LIN {X -0.118,Y -195.849,Z 1330.705,A 0.000,B 0.000,C 90.000,E1 126.870} C_DIS
LIN {X 0.022,Y -199.211,Z 1330.695,A 0.000,B 0.000,C 90.000,E1 125.105} C_DIS
LIN {X -0.016,Y -309.077,Z 1330.695,A 0.000,B 0.000,C 90.000,E1 125.105} C_DIS
LIN {X -0.170,Y -310.750,Z 1330.695,A 0.000,B 0.000,C 90.000,E1 125.105} C_DIS
LIN {X 0.024,Y -314.683,Z 1330.694,A 0.000,B 0.000,C 90.000,E1 124.898} C_DIS
LIN {X -0.037,Y -316.948,Z 1330.693,A 0.000,B 0.000,C 90.000,E1 124.739} C_DIS
LIN {X -0.082,Y -320.065,Z 1330.691,A 0.000,B 0.000,C 90.000,E1 124.405} C_DIS
LIN {X -0.155,Y -322.032,Z 1330.689,A 0.000,B 0.000,C 90.000,E1 124.119} C_DIS
LIN {X 0.038,Y -323.567,Z 1330.688,A 0.000,B 0.000,C 90.000,E1 123.785} C_DIS
LIN {X -0.056,Y -325.946,Z 1330.684,A 0.000,B 0.000,C 90.000,E1 123.166} C_DIS
LIN {X -0.055,Y -336.432,Z 1330.668,A 0.000,B 0.000,C 90.000,E1 120.335} C_DIS
LIN {X 0.200,Y -348.268,Z 1330.653,A 0.000,B 0.000,C 90.000,E1 117.513} C_DIS
LIN {X 0.001,Y -361.549,Z 1330.638,A 0.000,B 0.000,C 90.000,E1 114.823} C_DIS
LIN {X -0.050,Y -374.665,Z 1330.625,A 0.000,B 0.000,C 90.000,E1 112.461} C_DIS
LIN {X 0.093,Y -389.108,Z 1330.612,A 0.000,B 0.000,C 90.000,E1 110.120} C_DIS
LIN {X -0.043,Y -404.981,Z 1330.599,A 0.000,B 0.000,C 90.000,E1 107.873} C_DIS
LIN {X -0.042,Y -422.391,Z 1330.587,A 0.000,B 0.000,C 90.000,E1 105.662} C_DIS
LIN {X -0.232,Y -441.441,Z 1330.575,A 0.000,B 0.000,C 90.000,E1 103.536} C_DIS
LIN {X 0.089,Y -461.498,Z 1330.564,A 0.000,B 0.000,C 90.000,E1 101.478} C_DIS
LIN {X 0.089,Y -479.451,Z 1330.555,A 0.000,B 0.000,C 90.000,E1 99.849} C_DIS
LIN {X 0.151,Y -481.477,Z 1330.553,A 0.000,B 0.000,C 90.000,E1 99.613} C_DIS
LIN {X 0.212,Y -483.021,Z 1330.552,A 0.000,B 0.000,C 90.000,E1 99.378} C_DIS
LIN {X 0.017,Y -484.300,Z 1330.551,A 0.000,B 0.000,C 90.000,E1 99.151} C_DIS
LIN {X -0.100,Y -485.240,Z 1330.549,A 0.000,B 0.000,C 90.000,E1 98.916} C_DIS
LIN {X 0.086,Y -486.268,Z 1330.547,A 0.000,B 0.000,C 90.000,E1 98.398} C_DIS
LIN {X -0.202,Y -486.295,Z 1330.544,A 0.000,B 0.000,C 90.000,E1 97.936} C_DIS
LIN {X 0.062,Y -485.327,Z 1330.541,A 0.000,B 0.000,C 90.000,E1 97.409} C_DIS
LIN {X -0.220,Y -483.199,Z 1330.538,A 0.000,B 0.000,C 90.000,E1 96.947} C_DIS
LIN {X 0.088,Y -481.557,Z 1330.537,A 0.000,B 0.000,C 90.000,E1 96.663} C_DIS
LIN {X 0.091,Y -470.630,Z 1330.529,A 0.000,B 0.000,C 90.000,E1 95.163} C_DIS
LIN {X -0.105,Y -457.075,Z 1330.517,A 0.000,B 0.000,C 90.000,E1 93.154} C_DIS
LIN {X 0.043,Y -442.213,Z 1330.505,A 0.000,B 0.000,C 90.000,E1 90.802} C_DIS
LIN {X 0.074,Y -425.766,Z 1330.488,A 0.000,B 0.000,C 90.000,E1 87.879} C_DIS
LIN {X 0.057,Y -415.709,Z 1330.478,A 0.000,B 0.000,C 90.000,E1 85.988} C_DIS
LIN {X -0.119,Y -405.430,Z 1330.467,A 0.000,B 0.000,C 90.000,E1 84.090} C_DIS
LIN {X -0.079,Y -396.463,Z 1330.458,A 0.000,B 0.000,C 90.000,E1 82.413} C_DIS
LIN {X -0.194,Y -387.225,Z 1330.448,A 0.000,B 0.000,C 90.000,E1 80.735} C_DIS
LIN {X -0.039,Y -377.786,Z 1330.439,A 0.000,B 0.000,C 90.000,E1 78.993} C_DIS
LIN {X 0.079,Y -366.465,Z 1330.427,A 0.000,B 0.000,C 90.000,E1 76.937} C_DIS
LIN {X 0.042,Y -354.979,Z 1330.416,A 0.000,B 0.000,C 90.000,E1 74.866} C_DIS
LIN {X -0.132,Y -343.438,Z 1330.404,A 0.000,B 0.000,C 90.000,E1 72.779} C_DIS
LIN {X -0.041,Y -330.180,Z 1330.391,A 0.000,B 0.000,C 90.000,E1 70.296} C_DIS
LIN {X -0.165,Y -317.253,Z 1330.376,A 0.000,B 0.000,C 90.000,E1 67.794} C_DIS
LIN {X -0.017,Y -300.759,Z 1330.357,A 0.000,B 0.000,C 90.000,E1 64.204} C_DIS
LIN {X -0.088,Y -291.482,Z 1330.344,A 0.000,B 0.000,C 90.000,E1 61.897} C_DIS
LIN {X -0.060,Y -284.436,Z 1330.333,A 0.000,B 0.000,C 90.000,E1 59.871} C_DIS
LIN {X 0.090,Y -274.075,Z 1330.314,A 0.000,B 0.000,C 90.000,E1 56.421} C_DIS
LIN {X -0.062,Y -264.729,Z 1330.294,A 0.000,B 0.000,C 90.000,E1 52.970} C_DIS
LIN {X 0.136,Y -255.963,Z 1330.275,A 0.000,B 0.000,C 90.000,E1 49.380} C_DIS
LIN {X -0.041,Y -249.331,Z 1330.259,A 0.000,B 0.000,C 90.000,E1 46.539} C_DIS
LIN {X 0.104,Y -241.390,Z 1330.238,A 0.000,B 0.000,C 90.000,E1 42.852} C_DIS
LIN {X -0.129,Y -234.080,Z 1330.218,A 0.000,B 0.000,C 90.000,E1 39.197} C_DIS
LIN {X 0.032,Y -227.630,Z 1330.197,A 0.000,B 0.000,C 90.000,E1 35.391} C_DIS
LIN {X -0.031,Y -222.216,Z 1330.175,A 0.000,B 0.000,C 90.000,E1 31.592} C_DIS
LIN {X 0.009,Y -217.022,Z 1330.150,A 0.000,B 0.000,C 90.000,E1 26.950} C_DIS
LIN {X -0.033,Y -212.863,Z 1330.124,A 0.000,B 0.000,C 90.000,E1 22.280} C_DIS
LIN {X -0.082,Y -209.866,Z 1330.102,A 0.000,B 0.000,C 90.000,E1 18.362} C_DIS
LIN {X -0.046,Y -207.669,Z 1330.084,A 0.000,B 0.000,C 90.000,E1 15.190} C_DIS
LIN {X -0.028,Y -205.583,Z 1330.067,A 0.000,B 0.000,C 90.000,E1 12.007} C_DIS
LIN {X -0.090,Y -202.497,Z 1330.036,A 0.000,B 0.000,C 90.000,E1 6.429} C_DIS
LIN {X 0.000,Y -200.364,Z 1330.000,A 0.000,B 0.000,C 90.000,E1 360.000} C_DIS
LIN {X 0.070,Y -200.097,Z 1329.962,A 0.000,B 0.000,C 90.000,E1 353.053} C_DIS
LIN {X -0.087,Y -201.859,Z 1329.926,A 0.000,B 0.000,C 90.000,E1 346.645} C_DIS
LIN {X 0.053,Y -205.124,Z 1329.894,A 0.000,B 0.000,C 90.000,E1 340.986} C_DIS
LIN {X -0.036,Y -209.391,Z 1329.868,A 0.000,B 0.000,C 90.000,E1 336.230} C_DIS
LIN {X -0.037,Y -213.991,Z 1329.846,A 0.000,B 0.000,C 90.000,E1 332.281} C_DIS
LIN {X 0.135,Y -219.620,Z 1329.824,A 0.000,B 0.000,C 90.000,E1 328.329} C_DIS
LIN {X 0.086,Y -226.283,Z 1329.803,A 0.000,B 0.000,C 90.000,E1 324.482} C_DIS
LIN {X -0.004,Y -232.326,Z 1329.786,A 0.000,B 0.000,C 90.000,E1 321.457} C_DIS
LIN {X -0.064,Y -240.993,Z 1329.765,A 0.000,B 0.000,C 90.000,E1 317.715} C_DIS
LIN {X 0.112,Y -249.732,Z 1329.747,A 0.000,B 0.000,C 90.000,E1 314.352} C_DIS
LIN {X 0.033,Y -258.740,Z 1329.730,A 0.000,B 0.000,C 90.000,E1 311.472} C_DIS
LIN {X -0.027,Y -267.675,Z 1329.717,A 0.000,B 0.000,C 90.000,E1 308.991} C_DIS
LIN {X 0.091,Y -279.387,Z 1329.701,A 0.000,B 0.000,C 90.000,E1 306.171} C_DIS
LIN {X 0.074,Y -289.324,Z 1329.690,A 0.000,B 0.000,C 90.000,E1 304.119} C_DIS
LIN {X -0.087,Y -298.444,Z 1329.680,A 0.000,B 0.000,C 90.000,E1 302.467} C_DIS
LIN {X -0.017,Y -308.572,Z 1329.671,A 0.000,B 0.000,C 90.000,E1 300.797} C_DIS
LIN {X 0.008,Y -317.490,Z 1329.664,A 0.000,B 0.000,C 90.000,E1 299.489} C_DIS
LIN {X -0.020,Y -329.613,Z 1329.655,A 0.000,B 0.000,C 90.000,E1 297.897} C_DIS
LIN {X 0.065,Y -350.580,Z 1329.641,A 0.000,B 0.000,C 90.000,E1 295.412} C_DIS
LIN {X -0.084,Y -363.624,Z 1329.633,A 0.000,B 0.000,C 90.000,E1 293.951} C_DIS
LIN {X 0.018,Y -373.873,Z 1329.626,A 0.000,B 0.000,C 90.000,E1 292.770} C_DIS
LIN {X 0.120,Y -383.899,Z 1329.620,A 0.000,B 0.000,C 90.000,E1 291.589} C_DIS
LIN {X -0.166,Y -400.941,Z 1329.609,A 0.000,B 0.000,C 90.000,E1 289.631} C_DIS
LIN {X -0.083,Y -415.751,Z 1329.600,A 0.000,B 0.000,C 90.000,E1 287.946} C_DIS
LIN {X -0.142,Y -425.351,Z 1329.594,A 0.000,B 0.000,C 90.000,E1 286.858} C_DIS
LIN {X 0.029,Y -432.158,Z 1329.589,A 0.000,B 0.000,C 90.000,E1 286.024} C_DIS
LIN {X -0.149,Y -438.442,Z 1329.585,A 0.000,B 0.000,C 90.000,E1 285.245} C_DIS
LIN {X 0.034,Y -444.085,Z 1329.580,A 0.000,B 0.000,C 90.000,E1 284.426} C_DIS
LIN {X -0.044,Y -449.062,Z 1329.576,A 0.000,B 0.000,C 90.000,E1 283.647} C_DIS
LIN {X -0.196,Y -453.340,Z 1329.571,A 0.000,B 0.000,C 90.000,E1 282.883} C_DIS
LIN {X 0.140,Y -456.820,Z 1329.567,A 0.000,B 0.000,C 90.000,E1 282.063} C_DIS
LIN {X -0.041,Y -457.839,Z 1329.566,A 0.000,B 0.000,C 90.000,E1 281.827} C_DIS
LIN {X 0.057,Y -459.565,Z 1329.563,A 0.000,B 0.000,C 90.000,E1 281.299} C_DIS
LIN {X 0.074,Y -460.955,Z 1329.560,A 0.000,B 0.000,C 90.000,E1 280.782} C_DIS
LIN {X 0.189,Y -461.962,Z 1329.557,A 0.000,B 0.000,C 90.000,E1 280.254} C_DIS
LIN {X -0.146,Y -462.526,Z 1329.554,A 0.000,B 0.000,C 90.000,E1 279.782} C_DIS
LIN {X -0.099,Y -462.700,Z 1329.551,A 0.000,B 0.000,C 90.000,E1 279.265} C_DIS
LIN {X -0.044,Y -462.433,Z 1329.549,A 0.000,B 0.000,C 90.000,E1 278.746} C_DIS
LIN {X 0.080,Y -461.733,Z 1329.546,A 0.000,B 0.000,C 90.000,E1 278.219} C_DIS
LIN {X 0.135,Y -460.499,Z 1329.543,A 0.000,B 0.000,C 90.000,E1 277.701} C_DIS
LIN {X 0.011,Y -457.672,Z 1329.539,A 0.000,B 0.000,C 90.000,E1 276.947} C_DIS
LIN {X 0.047,Y -455.107,Z 1329.536,A 0.000,B 0.000,C 90.000,E1 276.429} C_DIS
LIN {X -0.189,Y -453.660,Z 1329.534,A 0.000,B 0.000,C 90.000,E1 276.201} C_DIS
LIN {X -0.173,Y -450.230,Z 1329.531,A 0.000,B 0.000,C 90.000,E1 275.682} C_DIS
LIN {X -0.175,Y -446.094,Z 1329.529,A 0.000,B 0.000,C 90.000,E1 275.163} C_DIS
LIN {X 0.015,Y -443.722,Z 1329.527,A 0.000,B 0.000,C 90.000,E1 274.878} C_DIS
LIN {X 0.079,Y -438.319,Z 1329.524,A 0.000,B 0.000,C 90.000,E1 274.359} C_DIS
LIN {X -0.025,Y -432.416,Z 1329.522,A 0.000,B 0.000,C 90.000,E1 273.898} C_DIS
LIN {X -0.196,Y -426.155,Z 1329.519,A 0.000,B 0.000,C 90.000,E1 273.498} C_DIS
LIN {X 0.037,Y -419.659,Z 1329.517,A 0.000,B 0.000,C 90.000,E1 273.094} C_DIS
LIN {X 0.156,Y -413.002,Z 1329.515,A 0.000,B 0.000,C 90.000,E1 272.751} C_DIS
LIN {X 0.139,Y -406.290,Z 1329.514,A 0.000,B 0.000,C 90.000,E1 272.465} C_DIS
LIN {X -0.014,Y -399.093,Z 1329.512,A 0.000,B 0.000,C 90.000,E1 272.236} C_DIS
LIN {X 0.119,Y -391.578,Z 1329.511,A 0.000,B 0.000,C 90.000,E1 272.007} C_DIS
LIN {X 0.130,Y -383.979,Z 1329.510,A 0.000,B 0.000,C 90.000,E1 271.835} C_DIS
LIN {X -0.002,Y -376.274,Z 1329.510,A 0.000,B 0.000,C 90.000,E1 271.718} C_DIS
LIN {X 0.034,Y -367.410,Z 1329.509,A 0.000,B 0.000,C 90.000,E1 271.604} C_DIS
LIN {X -0.025,Y -358.395,Z 1329.509,A 0.000,B 0.000,C 90.000,E1 271.547} C_DIS
LIN {X 0.157,Y -350.749,Z 1329.508,A 0.000,B 0.000,C 90.000,E1 271.489} C_DIS
LIN {X 0.052,Y -181.350,Z 1329.508,A 0.000,B 0.000,C 90.000,E1 271.489} C_DIS
LIN {X -0.083,Y -181.556,Z 1329.500,A 0.000,B 0.000,C 90.000,E1 270.000} C_DIS
LIN {X 0.054,Y -180.901,Z 1329.474,A 0.000,B 0.000,C 90.000,E1 265.241} C_DIS
LIN {X 0.003,Y -180.225,Z 1329.464,A 0.000,B 0.000,C 90.000,E1 263.571} C_DIS
LIN {X -0.044,Y -179.040,Z 1329.446,A 0.000,B 0.000,C 90.000,E1 260.208} C_DIS
LIN {X 0.020,Y -178.707,Z 1329.441,A 0.000,B 0.000,C 90.000,E1 259.342} C_DIS
LIN {X -0.039,Y -175.755,Z 1329.412,A 0.000,B 0.000,C 90.000,E1 254.267} C_DIS
LIN {X -0.037,Y -171.938,Z 1329.384,A 0.000,B 0.000,C 90.000,E1 249.135} C_DIS
LIN {X -0.061,Y -171.321,Z 1329.379,A 0.000,B 0.000,C 90.000,E1 248.284} C_DIS
LIN {X -0.008,Y -167.578,Z 1329.355,A 0.000,B 0.000,C 90.000,E1 243.948} C_DIS
LIN {X -0.068,Y -166.211,Z 1329.346,A 0.000,B 0.000,C 90.000,E1 242.231} C_DIS
LIN {X -0.080,Y -162.975,Z 1329.326,A 0.000,B 0.000,C 90.000,E1 238.742} C_DIS
LIN {X -0.032,Y -160.889,Z 1329.312,A 0.000,B 0.000,C 90.000,E1 236.087} C_DIS
LIN {X -0.054,Y -157.658,Z 1329.292,A 0.000,B 0.000,C 90.000,E1 232.557} C_DIS
LIN {X 0.004,Y -155.696,Z 1329.277,A 0.000,B 0.000,C 90.000,E1 229.865} C_DIS
LIN {X -0.060,Y -151.960,Z 1329.252,A 0.000,B 0.000,C 90.000,E1 225.405} C_DIS
LIN {X -0.043,Y -150.201,Z 1329.237,A 0.000,B 0.000,C 90.000,E1 222.690} C_DIS
LIN {X 0.088,Y -146.969,Z 1329.212,A 0.000,B 0.000,C 90.000,E1 218.096} C_DIS
LIN {X -0.009,Y -145.556,Z 1329.197,A 0.000,B 0.000,C 90.000,E1 215.391} C_DIS
LIN {X -0.010,Y -142.950,Z 1329.171,A 0.000,B 0.000,C 90.000,E1 210.797} C_DIS
LIN {X 0.048,Y -141.575,Z 1329.151,A 0.000,B 0.000,C 90.000,E1 207.078} C_DIS
LIN {X -0.031,Y -139.414,Z 1329.114,A 0.000,B 0.000,C 90.000,E1 200.610} C_DIS
LIN {X 0.022,Y -139.137,Z 1329.104,A 0.000,B 0.000,C 90.000,E1 198.725} C_DIS
LIN {X 0.048,Y -138.348,Z 1329.057,A 0.000,B 0.000,C 90.000,E1 190.310} C_DIS
LIN {X 0.036,Y -139.494,Z 1329.005,A 0.000,B 0.000,C 90.000,E1 180.974} C_DIS
LIN {X -0.023,Y -141.108,Z 1328.974,A 0.000,B 0.000,C 90.000,E1 175.412} C_DIS
LIN {X -0.069,Y -142.486,Z 1328.959,A 0.000,B 0.000,C 90.000,E1 172.648} C_DIS
LIN {X 0.019,Y -144.738,Z 1328.933,A 0.000,B 0.000,C 90.000,E1 167.993} C_DIS
LIN {X -0.031,Y -147.343,Z 1328.913,A 0.000,B 0.000,C 90.000,E1 164.338} C_DIS
LIN {X 0.034,Y -150.668,Z 1328.888,A 0.000,B 0.000,C 90.000,E1 159.752} C_DIS
LIN {X -0.086,Y -154.147,Z 1328.867,A 0.000,B 0.000,C 90.000,E1 156.177} C_DIS
LIN {X 0.049,Y -157.577,Z 1328.848,A 0.000,B 0.000,C 90.000,E1 152.538} C_DIS
LIN {X 0.000,Y -161.823,Z 1328.828,A 0.000,B 0.000,C 90.000,E1 148.997} C_DIS
LIN {X 0.019,Y -166.013,Z 1328.808,A 0.000,B 0.000,C 90.000,E1 145.468} C_DIS
LIN {X 0.012,Y -171.014,Z 1328.789,A 0.000,B 0.000,C 90.000,E1 141.984} C_DIS
LIN {X 0.043,Y -175.884,Z 1328.770,A 0.000,B 0.000,C 90.000,E1 138.528} C_DIS
LIN {X -0.081,Y -181.488,Z 1328.751,A 0.000,B 0.000,C 90.000,E1 135.162} C_DIS
LIN {X 0.055,Y -187.004,Z 1328.732,A 0.000,B 0.000,C 90.000,E1 131.757} C_DIS
LIN {X 0.057,Y -190.121,Z 1328.723,A 0.000,B 0.000,C 90.000,E1 130.092} C_DIS
LIN {X 0.077,Y -195.892,Z 1328.704,A 0.000,B 0.000,C 90.000,E1 126.790} C_DIS
LIN {X 0.010,Y -199.218,Z 1328.695,A 0.000,B 0.000,C 90.000,E1 125.105} C_DIS
LIN {X -0.019,Y -308.719,Z 1328.695,A 0.000,B 0.000,C 90.000,E1 125.105} C_DIS
LIN {X 0.138,Y -311.452,Z 1328.695,A 0.000,B 0.000,C 90.000,E1 125.025} C_DIS
LIN {X 0.096,Y -317.160,Z 1328.693,A 0.000,B 0.000,C 90.000,E1 124.692} C_DIS
LIN {X 0.053,Y -320.203,Z 1328.691,A 0.000,B 0.000,C 90.000,E1 124.358} C_DIS
LIN {X -0.048,Y -322.166,Z 1328.689,A 0.000,B 0.000,C 90.000,E1 124.072} C_DIS
LIN {X -0.151,Y -323.693,Z 1328.688,A 0.000,B 0.000,C 90.000,E1 123.785} C_DIS
LIN {X 0.030,Y -327.143,Z 1328.682,A 0.000,B 0.000,C 90.000,E1 122.801} C_DIS
LIN {X -0.118,Y -337.791,Z 1328.667,A 0.000,B 0.000,C 90.000,E1 120.001} C_DIS
LIN {X 0.017,Y -349.795,Z 1328.651,A 0.000,B 0.000,C 90.000,E1 117.206} C_DIS
LIN {X -0.143,Y -363.265,Z 1328.636,A 0.000,B 0.000,C 90.000,E1 114.515} C_DIS
LIN {X -0.153,Y -376.560,Z 1328.623,A 0.000,B 0.000,C 90.000,E1 112.153} C_DIS
LIN {X 0.034,Y -391.195,Z 1328.610,A 0.000,B 0.000,C 90.000,E1 109.812} C_DIS
LIN {X -0.181,Y -407.272,Z 1328.598,A 0.000,B 0.000,C 90.000,E1 107.583} C_DIS
LIN {X -0.121,Y -424.906,Z 1328.585,A 0.000,B 0.000,C 90.000,E1 105.371} C_DIS
LIN {X -0.124,Y -444.169,Z 1328.573,A 0.000,B 0.000,C 90.000,E1 103.231} C_DIS
LIN {X -0.164,Y -464.307,Z 1328.562,A 0.000,B 0.000,C 90.000,E1 101.243} C_DIS
LIN {X -0.115,Y -479.654,Z 1328.555,A 0.000,B 0.000,C 90.000,E1 99.849} C_DIS
LIN {X -0.077,Y -481.619,Z 1328.553,A 0.000,B 0.000,C 90.000,E1 99.613} C_DIS
LIN {X -0.041,Y -483.117,Z 1328.552,A 0.000,B 0.000,C 90.000,E1 99.378} C_DIS
LIN {X -0.234,Y -484.341,Z 1328.551,A 0.000,B 0.000,C 90.000,E1 99.151} C_DIS
LIN {X 0.127,Y -485.233,Z 1328.549,A 0.000,B 0.000,C 90.000,E1 98.859} C_DIS
LIN {X -0.166,Y -486.182,Z 1328.547,A 0.000,B 0.000,C 90.000,E1 98.398} C_DIS
LIN {X 0.094,Y -486.137,Z 1328.544,A 0.000,B 0.000,C 90.000,E1 97.871} C_DIS
LIN {X -0.190,Y -485.092,Z 1328.541,A 0.000,B 0.000,C 90.000,E1 97.409} C_DIS
LIN {X 0.119,Y -484.146,Z 1328.540,A 0.000,B 0.000,C 90.000,E1 97.125} C_DIS
LIN {X 0.008,Y -482.863,Z 1328.538,A 0.000,B 0.000,C 90.000,E1 96.891} C_DIS
LIN {X 0.012,Y -477.362,Z 1328.534,A 0.000,B 0.000,C 90.000,E1 96.144} C_DIS
LIN {X 0.071,Y -460.015,Z 1328.520,A 0.000,B 0.000,C 90.000,E1 93.612} C_DIS
LIN {X -0.219,Y -441.790,Z 1328.504,A 0.000,B 0.000,C 90.000,E1 90.802} C_DIS
LIN {X -0.191,Y -425.367,Z 1328.488,A 0.000,B 0.000,C 90.000,E1 87.879} C_DIS
LIN {X -0.210,Y -415.310,Z 1328.478,A 0.000,B 0.000,C 90.000,E1 85.988} C_DIS
LIN {X 0.015,Y -405.047,Z 1328.467,A 0.000,B 0.000,C 90.000,E1 84.033} C_DIS
LIN {X 0.045,Y -396.053,Z 1328.458,A 0.000,B 0.000,C 90.000,E1 82.356} C_DIS
LIN {X -0.082,Y -386.831,Z 1328.448,A 0.000,B 0.000,C 90.000,E1 80.679} C_DIS
LIN {X 0.133,Y -377.393,Z 1328.439,A 0.000,B 0.000,C 90.000,E1 78.926} C_DIS
LIN {X 0.173,Y -367.681,Z 1328.429,A 0.000,B 0.000,C 90.000,E1 77.173} C_DIS
LIN {X 0.072,Y -356.206,Z 1328.417,A 0.000,B 0.000,C 90.000,E1 75.117} C_DIS
LIN {X -0.011,Y -346.314,Z 1328.407,A 0.000,B 0.000,C 90.000,E1 73.323} C_DIS
LIN {X 0.044,Y -334.690,Z 1328.395,A 0.000,B 0.000,C 90.000,E1 71.167} C_DIS
LIN {X 0.132,Y -321.650,Z 1328.381,A 0.000,B 0.000,C 90.000,E1 68.646} C_DIS
LIN {X 0.172,Y -304.722,Z 1328.362,A 0.000,B 0.000,C 90.000,E1 65.101} C_DIS
LIN {X 0.166,Y -296.337,Z 1328.351,A 0.000,B 0.000,C 90.000,E1 63.127} C_DIS
LIN {X -0.115,Y -288.758,Z 1328.340,A 0.000,B 0.000,C 90.000,E1 61.179} C_DIS
LIN {X 0.006,Y -282.017,Z 1328.328,A 0.000,B 0.000,C 90.000,E1 59.125} C_DIS
LIN {X 0.088,Y -271.923,Z 1328.309,A 0.000,B 0.000,C 90.000,E1 55.674} C_DIS
LIN {X 0.022,Y -262.762,Z 1328.290,A 0.000,B 0.000,C 90.000,E1 52.190} C_DIS
LIN {X -0.050,Y -254.151,Z 1328.270,A 0.000,B 0.000,C 90.000,E1 48.647} C_DIS
LIN {X 0.069,Y -247.580,Z 1328.254,A 0.000,B 0.000,C 90.000,E1 45.729} C_DIS
LIN {X -0.007,Y -239.763,Z 1328.234,A 0.000,B 0.000,C 90.000,E1 42.081} C_DIS
LIN {X -0.109,Y -232.592,Z 1328.213,A 0.000,B 0.000,C 90.000,E1 38.382} C_DIS
LIN {X -0.131,Y -226.361,Z 1328.192,A 0.000,B 0.000,C 90.000,E1 34.612} C_DIS
LIN {X 0.025,Y -221.164,Z 1328.171,A 0.000,B 0.000,C 90.000,E1 30.747} C_DIS
LIN {X 0.031,Y -216.198,Z 1328.145,A 0.000,B 0.000,C 90.000,E1 26.104} C_DIS
LIN {X 0.058,Y -212.128,Z 1328.119,A 0.000,B 0.000,C 90.000,E1 21.408} C_DIS
LIN {X 0.107,Y -209.153,Z 1328.097,A 0.000,B 0.000,C 90.000,E1 17.457} C_DIS
LIN {X 0.063,Y -206.968,Z 1328.080,A 0.000,B 0.000,C 90.000,E1 14.300} C_DIS
LIN {X 0.095,Y -204.406,Z 1328.057,A 0.000,B 0.000,C 90.000,E1 10.310} C_DIS
LIN {X 0.072,Y -201.950,Z 1328.031,A 0.000,B 0.000,C 90.000,E1 5.511} C_DIS
LIN {X -0.054,Y -200.031,Z 1327.993,A 0.000,B 0.000,C 90.000,E1 358.740} C_DIS
LIN {X 0.072,Y -200.124,Z 1327.957,A 0.000,B 0.000,C 90.000,E1 352.243} C_DIS
LIN {X -0.095,Y -201.834,Z 1327.926,A 0.000,B 0.000,C 90.000,E1 346.645} C_DIS
LIN {X 0.044,Y -205.156,Z 1327.894,A 0.000,B 0.000,C 90.000,E1 340.986} C_DIS
LIN {X -0.043,Y -209.465,Z 1327.868,A 0.000,B 0.000,C 90.000,E1 336.230} C_DIS
LIN {X -0.042,Y -214.083,Z 1327.846,A 0.000,B 0.000,C 90.000,E1 332.281} C_DIS
LIN {X 0.133,Y -219.740,Z 1327.824,A 0.000,B 0.000,C 90.000,E1 328.329} C_DIS
LIN {X 0.088,Y -226.400,Z 1327.803,A 0.000,B 0.000,C 90.000,E1 324.482} C_DIS
LIN {X 0.001,Y -232.433,Z 1327.786,A 0.000,B 0.000,C 90.000,E1 321.457} C_DIS
LIN {X -0.055,Y -241.110,Z 1327.765,A 0.000,B 0.000,C 90.000,E1 317.715} C_DIS
LIN {X 0.123,Y -249.834,Z 1327.747,A 0.000,B 0.000,C 90.000,E1 314.352} C_DIS
LIN {X 0.047,Y -258.819,Z 1327.730,A 0.000,B 0.000,C 90.000,E1 311.472} C_DIS
LIN {X -0.011,Y -267.762,Z 1327.717,A 0.000,B 0.000,C 90.000,E1 308.991} C_DIS
LIN {X 0.012,Y -277.912,Z 1327.703,A 0.000,B 0.000,C 90.000,E1 306.537} C_DIS
LIN {X -0.032,Y -287.698,Z 1327.692,A 0.000,B 0.000,C 90.000,E1 304.485} C_DIS
LIN {X -0.062,Y -298.540,Z 1327.680,A 0.000,B 0.000,C 90.000,E1 302.467} C_DIS
LIN {X 0.011,Y -308.668,Z 1327.671,A 0.000,B 0.000,C 90.000,E1 300.797} C_DIS
LIN {X 0.105,Y -319.931,Z 1327.662,A 0.000,B 0.000,C 90.000,E1 299.155} C_DIS
LIN {X -0.063,Y -332.281,Z 1327.653,A 0.000,B 0.000,C 90.000,E1 297.590} C_DIS
LIN {X 0.051,Y -350.692,Z 1327.641,A 0.000,B 0.000,C 90.000,E1 295.412} C_DIS
LIN {X -0.138,Y -363.761,Z 1327.633,A 0.000,B 0.000,C 90.000,E1 293.951} C_DIS
LIN {X -0.043,Y -373.998,Z 1327.626,A 0.000,B 0.000,C 90.000,E1 292.770} C_DIS
LIN {X 0.182,Y -386.436,Z 1327.618,A 0.000,B 0.000,C 90.000,E1 291.280} C_DIS
LIN {X -0.058,Y -403.492,Z 1327.607,A 0.000,B 0.000,C 90.000,E1 289.322} C_DIS
LIN {X -0.160,Y -415.865,Z 1327.600,A 0.000,B 0.000,C 90.000,E1 287.946} C_DIS
LIN {X -0.219,Y -425.466,Z 1327.594,A 0.000,B 0.000,C 90.000,E1 286.858} C_DIS
LIN {X -0.048,Y -432.286,Z 1327.589,A 0.000,B 0.000,C 90.000,E1 286.024} C_DIS
LIN {X 0.197,Y -438.554,Z 1327.584,A 0.000,B 0.000,C 90.000,E1 285.190} C_DIS
LIN {X -0.043,Y -444.208,Z 1327.580,A 0.000,B 0.000,C 90.000,E1 284.426} C_DIS
LIN {X -0.122,Y -449.160,Z 1327.576,A 0.000,B 0.000,C 90.000,E1 283.647} C_DIS
LIN {X 0.169,Y -453.421,Z 1327.571,A 0.000,B 0.000,C 90.000,E1 282.827} C_DIS
LIN {X 0.063,Y -456.942,Z 1327.567,A 0.000,B 0.000,C 90.000,E1 282.063} C_DIS
LIN {X -0.019,Y -459.703,Z 1327.563,A 0.000,B 0.000,C 90.000,E1 281.299} C_DIS
LIN {X -0.001,Y -461.100,Z 1327.560,A 0.000,B 0.000,C 90.000,E1 280.782} C_DIS
LIN {X 0.115,Y -462.077,Z 1327.557,A 0.000,B 0.000,C 90.000,E1 280.254} C_DIS
LIN {X 0.235,Y -462.695,Z 1327.554,A 0.000,B 0.000,C 90.000,E1 279.726} C_DIS
LIN {X -0.172,Y -462.915,Z 1327.551,A 0.000,B 0.000,C 90.000,E1 279.265} C_DIS
LIN {X -0.117,Y -462.663,Z 1327.548,A 0.000,B 0.000,C 90.000,E1 278.746} C_DIS
LIN {X 0.009,Y -461.961,Z 1327.546,A 0.000,B 0.000,C 90.000,E1 278.219} C_DIS
LIN {X 0.066,Y -460.740,Z 1327.543,A 0.000,B 0.000,C 90.000,E1 277.701} C_DIS
LIN {X -0.057,Y -457.970,Z 1327.539,A 0.000,B 0.000,C 90.000,E1 276.947} C_DIS
LIN {X -0.018,Y -455.455,Z 1327.536,A 0.000,B 0.000,C 90.000,E1 276.429} C_DIS
LIN {X 0.004,Y -452.354,Z 1327.533,A 0.000,B 0.000,C 90.000,E1 275.910} C_DIS
LIN {X 0.009,Y -448.614,Z 1327.530,A 0.000,B 0.000,C 90.000,E1 275.391} C_DIS
LIN {X 0.210,Y -446.543,Z 1327.529,A 0.000,B 0.000,C 90.000,E1 275.106} C_DIS
LIN {X 0.184,Y -441.563,Z 1327.526,A 0.000,B 0.000,C 90.000,E1 274.588} C_DIS
LIN {X 0.187,Y -435.734,Z 1327.523,A 0.000,B 0.000,C 90.000,E1 274.073} C_DIS
LIN {X -0.201,Y -429.621,Z 1327.520,A 0.000,B 0.000,C 90.000,E1 273.669} C_DIS
LIN {X -0.217,Y -423.154,Z 1327.518,A 0.000,B 0.000,C 90.000,E1 273.269} C_DIS
LIN {X 0.186,Y -416.575,Z 1327.516,A 0.000,B 0.000,C 90.000,E1 272.865} C_DIS
LIN {X 0.051,Y -409.861,Z 1327.514,A 0.000,B 0.000,C 90.000,E1 272.579} C_DIS
LIN {X -0.190,Y -403.104,Z 1327.513,A 0.000,B 0.000,C 90.000,E1 272.350} C_DIS
LIN {X 0.190,Y -395.765,Z 1327.512,A 0.000,B 0.000,C 90.000,E1 272.064} C_DIS
LIN {X -0.032,Y -384.629,Z 1327.510,A 0.000,B 0.000,C 90.000,E1 271.835} C_DIS
LIN {X -0.153,Y -376.913,Z 1327.509,A 0.000,B 0.000,C 90.000,E1 271.718} C_DIS
LIN {X -0.123,Y -368.238,Z 1327.509,A 0.000,B 0.000,C 90.000,E1 271.604} C_DIS
LIN {X 0.054,Y -355.147,Z 1327.508,A 0.000,B 0.000,C 90.000,E1 271.489} C_DIS
LIN {X -0.003,Y -352.126,Z 1327.508,A 0.000,B 0.000,C 90.000,E1 271.489} C_DIS
LIN {X -0.031,Y -181.355,Z 1327.508,A 0.000,B 0.000,C 90.000,E1 271.489} C_DIS
LIN {X 0.017,Y -181.552,Z 1327.500,A 0.000,B 0.000,C 90.000,E1 269.943} C_DIS
LIN {X -0.028,Y -180.899,Z 1327.474,A 0.000,B 0.000,C 90.000,E1 265.241} C_DIS
LIN {X -0.078,Y -180.213,Z 1327.464,A 0.000,B 0.000,C 90.000,E1 263.571} C_DIS
LIN {X 0.052,Y -179.034,Z 1327.445,A 0.000,B 0.000,C 90.000,E1 260.151} C_DIS
LIN {X -0.062,Y -178.689,Z 1327.441,A 0.000,B 0.000,C 90.000,E1 259.342} C_DIS
LIN {X 0.048,Y -175.739,Z 1327.412,A 0.000,B 0.000,C 90.000,E1 254.212} C_DIS
LIN {X 0.044,Y -171.922,Z 1327.384,A 0.000,B 0.000,C 90.000,E1 249.082} C_DIS
LIN {X 0.019,Y -171.295,Z 1327.379,A 0.000,B 0.000,C 90.000,E1 248.230} C_DIS
LIN {X 0.064,Y -167.558,Z 1327.355,A 0.000,B 0.000,C 90.000,E1 243.896} C_DIS
LIN {X 0.078,Y -166.182,Z 1327.345,A 0.000,B 0.000,C 90.000,E1 242.153} C_DIS
LIN {X 0.068,Y -162.953,Z 1327.326,A 0.000,B 0.000,C 90.000,E1 238.663} C_DIS
LIN {X -0.109,Y -160.861,Z 1327.311,A 0.000,B 0.000,C 90.000,E1 236.087} C_DIS
LIN {X 0.092,Y -157.636,Z 1327.292,A 0.000,B 0.000,C 90.000,E1 232.477} C_DIS
LIN {X 0.030,Y -155.673,Z 1327.277,A 0.000,B 0.000,C 90.000,E1 229.828} C_DIS
LIN {X 0.081,Y -151.940,Z 1327.252,A 0.000,B 0.000,C 90.000,E1 225.324} C_DIS
LIN {X 0.096,Y -150.178,Z 1327.237,A 0.000,B 0.000,C 90.000,E1 222.609} C_DIS
LIN {X 0.016,Y -146.953,Z 1327.212,A 0.000,B 0.000,C 90.000,E1 218.096} C_DIS
LIN {X 0.004,Y -145.541,Z 1327.196,A 0.000,B 0.000,C 90.000,E1 215.358} C_DIS
LIN {X -0.081,Y -142.936,Z 1327.171,A 0.000,B 0.000,C 90.000,E1 210.797} C_DIS
LIN {X -0.023,Y -141.560,Z 1327.150,A 0.000,B 0.000,C 90.000,E1 207.078} C_DIS
LIN {X 0.029,Y -139.409,Z 1327.114,A 0.000,B 0.000,C 90.000,E1 200.556} C_DIS
LIN {X -0.048,Y -139.129,Z 1327.104,A 0.000,B 0.000,C 90.000,E1 198.725} C_DIS
LIN {X -0.021,Y -138.350,Z 1327.057,A 0.000,B 0.000,C 90.000,E1 190.310} C_DIS
LIN {X -0.034,Y -139.498,Z 1327.005,A 0.000,B 0.000,C 90.000,E1 180.974} C_DIS
LIN {X 0.047,Y -141.120,Z 1326.974,A 0.000,B 0.000,C 90.000,E1 175.355} C_DIS
LIN {X 0.000,Y -142.500,Z 1326.959,A 0.000,B 0.000,C 90.000,E1 172.591} C_DIS
LIN {X -0.053,Y -144.755,Z 1326.933,A 0.000,B 0.000,C 90.000,E1 167.993} C_DIS
LIN {X 0.038,Y -147.365,Z 1326.913,A 0.000,B 0.000,C 90.000,E1 164.283} C_DIS
LIN {X -0.040,Y -150.692,Z 1326.887,A 0.000,B 0.000,C 90.000,E1 159.752} C_DIS
LIN {X 0.043,Y -154.171,Z 1326.867,A 0.000,B 0.000,C 90.000,E1 156.102} C_DIS
LIN {X -0.027,Y -157.606,Z 1326.847,A 0.000,B 0.000,C 90.000,E1 152.538} C_DIS
LIN {X -0.076,Y -161.858,Z 1326.828,A 0.000,B 0.000,C 90.000,E1 148.997} C_DIS
LIN {X -0.059,Y -166.049,Z 1326.808,A 0.000,B 0.000,C 90.000,E1 145.468} C_DIS
LIN {X -0.068,Y -171.053,Z 1326.789,A 0.000,B 0.000,C 90.000,E1 141.984} C_DIS
LIN {X -0.038,Y -175.925,Z 1326.770,A 0.000,B 0.000,C 90.000,E1 138.528} C_DIS
LIN {X -0.046,Y -180.164,Z 1326.755,A 0.000,B 0.000,C 90.000,E1 135.972} C_DIS
LIN {X -0.077,Y -185.581,Z 1326.737,A 0.000,B 0.000,C 90.000,E1 132.609} C_DIS
LIN {X -0.028,Y -190.171,Z 1326.723,A 0.000,B 0.000,C 90.000,E1 130.092} C_DIS
LIN {X 0.018,Y -197.500,Z 1326.700,A 0.000,B 0.000,C 90.000,E1 125.964} C_DIS
LIN {X 0.014,Y -199.216,Z 1326.695,A 0.000,B 0.000,C 90.000,E1 125.105} C_DIS
LIN {X -0.031,Y -308.256,Z 1326.695,A 0.000,B 0.000,C 90.000,E1 125.105} C_DIS
LIN {X -0.083,Y -309.516,Z 1326.695,A 0.000,B 0.000,C 90.000,E1 125.105} C_DIS
LIN {X 0.024,Y -314.551,Z 1326.694,A 0.000,B 0.000,C 90.000,E1 124.898} C_DIS
LIN {X -0.126,Y -317.031,Z 1326.693,A 0.000,B 0.000,C 90.000,E1 124.739} C_DIS
LIN {X 0.094,Y -320.349,Z 1326.691,A 0.000,B 0.000,C 90.000,E1 124.326} C_DIS
LIN {X -0.012,Y -322.280,Z 1326.689,A 0.000,B 0.000,C 90.000,E1 124.040} C_DIS
LIN {X 0.149,Y -323.785,Z 1326.687,A 0.000,B 0.000,C 90.000,E1 123.706} C_DIS
LIN {X -0.022,Y -328.334,Z 1326.680,A 0.000,B 0.000,C 90.000,E1 122.467} C_DIS
LIN {X -0.131,Y -339.139,Z 1326.665,A 0.000,B 0.000,C 90.000,E1 119.667} C_DIS
LIN {X 0.035,Y -351.316,Z 1326.649,A 0.000,B 0.000,C 90.000,E1 116.873} C_DIS
LIN {X 0.096,Y -364.966,Z 1326.634,A 0.000,B 0.000,C 90.000,E1 114.155} C_DIS
LIN {X -0.203,Y -378.436,Z 1326.621,A 0.000,B 0.000,C 90.000,E1 111.844} C_DIS
LIN {X 0.029,Y -393.260,Z 1326.608,A 0.000,B 0.000,C 90.000,E1 109.504} C_DIS
LIN {X -0.138,Y -409.540,Z 1326.596,A 0.000,B 0.000,C 90.000,E1 107.275} C_DIS
LIN {X -0.028,Y -427.393,Z 1326.584,A 0.000,B 0.000,C 90.000,E1 105.064} C_DIS
LIN {X -0.026,Y -446.827,Z 1326.572,A 0.000,B 0.000,C 90.000,E1 102.939} C_DIS
LIN {X 0.124,Y -467.041,Z 1326.561,A 0.000,B 0.000,C 90.000,E1 100.950} C_DIS
LIN {X 0.195,Y -479.794,Z 1326.555,A 0.000,B 0.000,C 90.000,E1 99.792} C_DIS
LIN {X 0.209,Y -481.716,Z 1326.553,A 0.000,B 0.000,C 90.000,E1 99.557} C_DIS
LIN {X 0.222,Y -483.179,Z 1326.552,A 0.000,B 0.000,C 90.000,E1 99.321} C_DIS
LIN {X -0.087,Y -485.207,Z 1326.549,A 0.000,B 0.000,C 90.000,E1 98.859} C_DIS
LIN {X 0.093,Y -486.088,Z 1326.546,A 0.000,B 0.000,C 90.000,E1 98.341} C_DIS
LIN {X -0.128,Y -485.976,Z 1326.544,A 0.000,B 0.000,C 90.000,E1 97.871} C_DIS
LIN {X 0.069,Y -484.858,Z 1326.541,A 0.000,B 0.000,C 90.000,E1 97.352} C_DIS
LIN {X -0.103,Y -483.872,Z 1326.540,A 0.000,B 0.000,C 90.000,E1 97.125} C_DIS
LIN {X -0.215,Y -482.536,Z 1326.538,A 0.000,B 0.000,C 90.000,E1 96.891} C_DIS
LIN {X -0.115,Y -468.103,Z 1326.527,A 0.000,B 0.000,C 90.000,E1 94.878} C_DIS
LIN {X 0.122,Y -454.548,Z 1326.516,A 0.000,B 0.000,C 90.000,E1 92.808} C_DIS
LIN {X -0.007,Y -441.395,Z 1326.504,A 0.000,B 0.000,C 90.000,E1 90.745} C_DIS
LIN {X 0.131,Y -423.568,Z 1326.486,A 0.000,B 0.000,C 90.000,E1 87.535} C_DIS
LIN {X 0.088,Y -413.465,Z 1326.476,A 0.000,B 0.000,C 90.000,E1 85.641} C_DIS
LIN {X -0.123,Y -403.184,Z 1326.465,A 0.000,B 0.000,C 90.000,E1 83.742} C_DIS
LIN {X -0.117,Y -394.170,Z 1326.456,A 0.000,B 0.000,C 90.000,E1 82.064} C_DIS
LIN {X 0.108,Y -384.914,Z 1326.446,A 0.000,B 0.000,C 90.000,E1 80.330} C_DIS
LIN {X -0.085,Y -375.394,Z 1326.437,A 0.000,B 0.000,C 90.000,E1 78.634} C_DIS
LIN {X -0.076,Y -365.665,Z 1326.427,A 0.000,B 0.000,C 90.000,E1 76.881} C_DIS
LIN {X -0.127,Y -354.173,Z 1326.416,A 0.000,B 0.000,C 90.000,E1 74.810} C_DIS
LIN {X 0.096,Y -344.268,Z 1326.405,A 0.000,B 0.000,C 90.000,E1 72.960} C_DIS
LIN {X -0.206,Y -332.650,Z 1326.393,A 0.000,B 0.000,C 90.000,E1 70.859} C_DIS
LIN {X 0.143,Y -319.683,Z 1326.380,A 0.000,B 0.000,C 90.000,E1 68.284} C_DIS
LIN {X -0.171,Y -302.935,Z 1326.360,A 0.000,B 0.000,C 90.000,E1 64.793} C_DIS
LIN {X 0.063,Y -293.438,Z 1326.347,A 0.000,B 0.000,C 90.000,E1 62.436} C_DIS
LIN {X -0.132,Y -286.171,Z 1326.336,A 0.000,B 0.000,C 90.000,E1 60.461} C_DIS
LIN {X -0.078,Y -275.642,Z 1326.317,A 0.000,B 0.000,C 90.000,E1 57.041} C_DIS
LIN {X 0.039,Y -266.191,Z 1326.297,A 0.000,B 0.000,C 90.000,E1 53.543} C_DIS
LIN {X 0.118,Y -257.382,Z 1326.278,A 0.000,B 0.000,C 90.000,E1 49.989} C_DIS
LIN {X -0.022,Y -250.733,Z 1326.262,A 0.000,B 0.000,C 90.000,E1 47.148} C_DIS
LIN {X -0.002,Y -242.718,Z 1326.242,A 0.000,B 0.000,C 90.000,E1 43.500} C_DIS
LIN {X -0.031,Y -235.231,Z 1326.221,A 0.000,B 0.000,C 90.000,E1 39.806} C_DIS
LIN {X 0.120,Y -228.624,Z 1326.200,A 0.000,B 0.000,C 90.000,E1 36.011} C_DIS
LIN {X 0.084,Y -223.038,Z 1326.179,A 0.000,B 0.000,C 90.000,E1 32.212} C_DIS
LIN {X 0.093,Y -218.439,Z 1326.158,A 0.000,B 0.000,C 90.000,E1 28.359} C_DIS
LIN {X 0.079,Y -213.976,Z 1326.132,A 0.000,B 0.000,C 90.000,E1 23.695} C_DIS
LIN {X -0.067,Y -210.748,Z 1326.110,A 0.000,B 0.000,C 90.000,E1 19.812} C_DIS
LIN {X 0.004,Y -207.872,Z 1326.088,A 0.000,B 0.000,C 90.000,E1 15.843} C_DIS
LIN {X 0.075,Y -205.717,Z 1326.070,A 0.000,B 0.000,C 90.000,E1 12.647} C_DIS
LIN {X 0.015,Y -202.885,Z 1326.044,A 0.000,B 0.000,C 90.000,E1 7.871} C_DIS
LIN {X 0.063,Y -200.873,Z 1326.017,A 0.000,B 0.000,C 90.000,E1 3.037} C_DIS
LIN {X 0.096,Y -199.757,Z 1325.979,A 0.000,B 0.000,C 90.000,E1 356.274} C_DIS
LIN {X -0.010,Y -201.166,Z 1325.935,A 0.000,B 0.000,C 90.000,E1 348.229} C_DIS
LIN {X -0.004,Y -204.018,Z 1325.903,A 0.000,B 0.000,C 90.000,E1 342.598} C_DIS
LIN {X 0.034,Y -207.918,Z 1325.877,A 0.000,B 0.000,C 90.000,E1 337.794} C_DIS
LIN {X -0.007,Y -212.203,Z 1325.855,A 0.000,B 0.000,C 90.000,E1 333.845} C_DIS
LIN {X -0.007,Y -217.451,Z 1325.833,A 0.000,B 0.000,C 90.000,E1 329.921} C_DIS
LIN {X 0.129,Y -223.740,Z 1325.811,A 0.000,B 0.000,C 90.000,E1 326.008} C_DIS
LIN {X 0.102,Y -230.950,Z 1325.790,A 0.000,B 0.000,C 90.000,E1 322.190} C_DIS
LIN {X 0.004,Y -239.381,Z 1325.769,A 0.000,B 0.000,C 90.000,E1 318.447} C_DIS
LIN {X -0.042,Y -248.902,Z 1325.749,A 0.000,B 0.000,C 90.000,E1 314.757} C_DIS
LIN {X 0.025,Y -257.717,Z 1325.732,A 0.000,B 0.000,C 90.000,E1 311.838} C_DIS
LIN {X -0.057,Y -266.490,Z 1325.719,A 0.000,B 0.000,C 90.000,E1 309.358} C_DIS
LIN {X 0.096,Y -276.453,Z 1325.705,A 0.000,B 0.000,C 90.000,E1 306.870} C_DIS
LIN {X 0.021,Y -286.081,Z 1325.693,A 0.000,B 0.000,C 90.000,E1 304.818} C_DIS
LIN {X -0.041,Y -296.741,Z 1325.682,A 0.000,B 0.000,C 90.000,E1 302.801} C_DIS
LIN {X 0.007,Y -306.641,Z 1325.673,A 0.000,B 0.000,C 90.000,E1 301.131} C_DIS
LIN {X 0.061,Y -317.671,Z 1325.664,A 0.000,B 0.000,C 90.000,E1 299.489} C_DIS
LIN {X -0.036,Y -332.356,Z 1325.653,A 0.000,B 0.000,C 90.000,E1 297.590} C_DIS
LIN {X 0.039,Y -350.763,Z 1325.641,A 0.000,B 0.000,C 90.000,E1 295.412} C_DIS
LIN {X -0.149,Y -363.833,Z 1325.633,A 0.000,B 0.000,C 90.000,E1 293.951} C_DIS
LIN {X -0.129,Y -374.147,Z 1325.626,A 0.000,B 0.000,C 90.000,E1 292.770} C_DIS
LIN {X 0.096,Y -386.564,Z 1325.618,A 0.000,B 0.000,C 90.000,E1 291.280} C_DIS
LIN {X -0.144,Y -403.607,Z 1325.607,A 0.000,B 0.000,C 90.000,E1 289.322} C_DIS
LIN {X -0.121,Y -416.005,Z 1325.599,A 0.000,B 0.000,C 90.000,E1 287.928} C_DIS
LIN {X 0.100,Y -425.604,Z 1325.593,A 0.000,B 0.000,C 90.000,E1 286.804} C_DIS
LIN {X -0.137,Y -432.423,Z 1325.589,A 0.000,B 0.000,C 90.000,E1 286.024} C_DIS
LIN {X 0.108,Y -438.672,Z 1325.584,A 0.000,B 0.000,C 90.000,E1 285.190} C_DIS
LIN {X -0.021,Y -444.296,Z 1325.580,A 0.000,B 0.000,C 90.000,E1 284.411} C_DIS
LIN {X 0.225,Y -449.253,Z 1325.576,A 0.000,B 0.000,C 90.000,E1 283.592} C_DIS
LIN {X 0.080,Y -453.484,Z 1325.571,A 0.000,B 0.000,C 90.000,E1 282.827} C_DIS
LIN {X -0.026,Y -456.988,Z 1325.567,A 0.000,B 0.000,C 90.000,E1 282.063} C_DIS
LIN {X -0.207,Y -458.040,Z 1325.566,A 0.000,B 0.000,C 90.000,E1 281.827} C_DIS
LIN {X -0.109,Y -459.813,Z 1325.563,A 0.000,B 0.000,C 90.000,E1 281.299} C_DIS
LIN {X -0.090,Y -461.226,Z 1325.560,A 0.000,B 0.000,C 90.000,E1 280.782} C_DIS
LIN {X 0.025,Y -462.252,Z 1325.557,A 0.000,B 0.000,C 90.000,E1 280.254} C_DIS
LIN {X 0.147,Y -462.873,Z 1325.554,A 0.000,B 0.000,C 90.000,E1 279.726} C_DIS
LIN {X 0.197,Y -463.068,Z 1325.551,A 0.000,B 0.000,C 90.000,E1 279.208} C_DIS
LIN {X -0.203,Y -462.831,Z 1325.548,A 0.000,B 0.000,C 90.000,E1 278.746} C_DIS
LIN {X -0.076,Y -462.156,Z 1325.546,A 0.000,B 0.000,C 90.000,E1 278.219} C_DIS
LIN {X -0.018,Y -460.951,Z 1325.543,A 0.000,B 0.000,C 90.000,E1 277.701} C_DIS
LIN {X 0.037,Y -459.269,Z 1325.540,A 0.000,B 0.000,C 90.000,E1 277.182} C_DIS
LIN {X 0.086,Y -457.034,Z 1325.537,A 0.000,B 0.000,C 90.000,E1 276.663} C_DIS
LIN {X 0.119,Y -454.336,Z 1325.534,A 0.000,B 0.000,C 90.000,E1 276.144} C_DIS
LIN {X 0.137,Y -450.952,Z 1325.531,A 0.000,B 0.000,C 90.000,E1 275.625} C_DIS
LIN {X 0.137,Y -446.929,Z 1325.528,A 0.000,B 0.000,C 90.000,E1 275.106} C_DIS
LIN {X 0.113,Y -442.057,Z 1325.526,A 0.000,B 0.000,C 90.000,E1 274.588} C_DIS
LIN {X 0.127,Y -436.331,Z 1325.523,A 0.000,B 0.000,C 90.000,E1 274.073} C_DIS
LIN {X 0.142,Y -430.247,Z 1325.520,A 0.000,B 0.000,C 90.000,E1 273.612} C_DIS
LIN {X 0.080,Y -423.833,Z 1325.518,A 0.000,B 0.000,C 90.000,E1 273.212} C_DIS
LIN {X 0.032,Y -417.183,Z 1325.516,A 0.000,B 0.000,C 90.000,E1 272.865} C_DIS
LIN {X 0.167,Y -407.240,Z 1325.514,A 0.000,B 0.000,C 90.000,E1 272.407} C_DIS
LIN {X 0.058,Y -400.352,Z 1325.512,A 0.000,B 0.000,C 90.000,E1 272.178} C_DIS
LIN {X -0.187,Y -393.000,Z 1325.511,A 0.000,B 0.000,C 90.000,E1 272.007} C_DIS
LIN {X -0.146,Y -385.599,Z 1325.510,A 0.000,B 0.000,C 90.000,E1 271.833} C_DIS
LIN {X 0.052,Y -373.568,Z 1325.509,A 0.000,B 0.000,C 90.000,E1 271.604} C_DIS
LIN {X 0.014,Y -360.126,Z 1325.508,A 0.000,B 0.000,C 90.000,E1 271.489} C_DIS
LIN {X 0.138,Y -349.086,Z 1325.508,A 0.000,B 0.000,C 90.000,E1 271.432} C_DIS
LIN {X 0.042,Y -181.362,Z 1325.508,A 0.000,B 0.000,C 90.000,E1 271.432} C_DIS
LIN {X -0.061,Y -181.547,Z 1325.500,A 0.000,B 0.000,C 90.000,E1 269.943} C_DIS
LIN {X 0.074,Y -180.896,Z 1325.473,A 0.000,B 0.000,C 90.000,E1 265.184} C_DIS
LIN {X -0.083,Y -179.842,Z 1325.459,A 0.000,B 0.000,C 90.000,E1 262.704} C_DIS
LIN {X -0.026,Y -179.027,Z 1325.445,A 0.000,B 0.000,C 90.000,E1 260.151} C_DIS
LIN {X 0.036,Y -178.673,Z 1325.441,A 0.000,B 0.000,C 90.000,E1 259.285} C_DIS
LIN {X -0.028,Y -175.724,Z 1325.412,A 0.000,B 0.000,C 90.000,E1 254.212} C_DIS
LIN {X -0.011,Y -172.440,Z 1325.389,A 0.000,B 0.000,C 90.000,E1 249.934} C_DIS
LIN {X -0.056,Y -171.270,Z 1325.379,A 0.000,B 0.000,C 90.000,E1 248.230} C_DIS
LIN {X -0.010,Y -167.540,Z 1325.355,A 0.000,B 0.000,C 90.000,E1 243.896} C_DIS
LIN {X 0.004,Y -166.157,Z 1325.345,A 0.000,B 0.000,C 90.000,E1 242.153} C_DIS
LIN {X -0.006,Y -162.932,Z 1325.326,A 0.000,B 0.000,C 90.000,E1 238.663} C_DIS
LIN {X -0.028,Y -161.603,Z 1325.316,A 0.000,B 0.000,C 90.000,E1 236.914} C_DIS
LIN {X -0.052,Y -159.129,Z 1325.301,A 0.000,B 0.000,C 90.000,E1 234.276} C_DIS
LIN {X -0.041,Y -155.650,Z 1325.277,A 0.000,B 0.000,C 90.000,E1 229.828} C_DIS
LIN {X 0.012,Y -151.922,Z 1325.252,A 0.000,B 0.000,C 90.000,E1 225.324} C_DIS
LIN {X 0.026,Y -150.156,Z 1325.237,A 0.000,B 0.000,C 90.000,E1 222.609} C_DIS
LIN {X -0.053,Y -146.937,Z 1325.212,A 0.000,B 0.000,C 90.000,E1 218.096} C_DIS
LIN {X 0.054,Y -145.525,Z 1325.196,A 0.000,B 0.000,C 90.000,E1 215.311} C_DIS
LIN {X 0.048,Y -142.924,Z 1325.171,A 0.000,B 0.000,C 90.000,E1 210.718} C_DIS
LIN {X -0.026,Y -141.547,Z 1325.150,A 0.000,B 0.000,C 90.000,E1 207.052} C_DIS
LIN {X -0.036,Y -139.404,Z 1325.114,A 0.000,B 0.000,C 90.000,E1 200.556} C_DIS
LIN {X 0.017,Y -139.122,Z 1325.104,A 0.000,B 0.000,C 90.000,E1 198.671} C_DIS
LIN {X 0.049,Y -138.351,Z 1325.057,A 0.000,B 0.000,C 90.000,E1 190.254} C_DIS
LIN {X 0.039,Y -139.502,Z 1325.005,A 0.000,B 0.000,C 90.000,E1 180.917} C_DIS
LIN {X -0.020,Y -141.131,Z 1324.974,A 0.000,B 0.000,C 90.000,E1 175.355} C_DIS
LIN {X -0.067,Y -142.512,Z 1324.959,A 0.000,B 0.000,C 90.000,E1 172.591} C_DIS
LIN {X 0.020,Y -144.771,Z 1324.933,A 0.000,B 0.000,C 90.000,E1 167.937} C_DIS
LIN {X -0.031,Y -147.385,Z 1324.913,A 0.000,B 0.000,C 90.000,E1 164.283} C_DIS
LIN {X 0.031,Y -150.714,Z 1324.887,A 0.000,B 0.000,C 90.000,E1 159.699} C_DIS
LIN {X -0.028,Y -154.195,Z 1324.867,A 0.000,B 0.000,C 90.000,E1 156.102} C_DIS
LIN {X 0.041,Y -157.635,Z 1324.847,A 0.000,B 0.000,C 90.000,E1 152.487} C_DIS
LIN {X -0.011,Y -161.892,Z 1324.828,A 0.000,B 0.000,C 90.000,E1 148.948} C_DIS
LIN {X 0.097,Y -166.082,Z 1324.808,A 0.000,B 0.000,C 90.000,E1 145.388} C_DIS
LIN {X 0.096,Y -171.090,Z 1324.789,A 0.000,B 0.000,C 90.000,E1 141.904} C_DIS
LIN {X 0.017,Y -175.963,Z 1324.769,A 0.000,B 0.000,C 90.000,E1 138.485} C_DIS
LIN {X -0.124,Y -180.207,Z 1324.755,A 0.000,B 0.000,C 90.000,E1 135.972} C_DIS
LIN {X 0.106,Y -185.623,Z 1324.736,A 0.000,B 0.000,C 90.000,E1 132.528} C_DIS
LIN {X -0.109,Y -190.219,Z 1324.723,A 0.000,B 0.000,C 90.000,E1 130.092} C_DIS
LIN {X 0.051,Y -197.546,Z 1324.700,A 0.000,B 0.000,C 90.000,E1 125.931} C_DIS
LIN {X -0.036,Y -199.245,Z 1324.695,A 0.000,B 0.000,C 90.000,E1 125.105} C_DIS
LIN {X -0.107,Y -309.463,Z 1324.695,A 0.000,B 0.000,C 90.000,E1 125.105} C_DIS
LIN {X -0.213,Y -310.545,Z 1324.695,A 0.000,B 0.000,C 90.000,E1 125.105} C_DIS
LIN {X -0.107,Y -314.844,Z 1324.694,A 0.000,B 0.000,C 90.000,E1 124.898} C_DIS
LIN {X 0.003,Y -317.233,Z 1324.693,A 0.000,B 0.000,C 90.000,E1 124.692} C_DIS
LIN {X -0.038,Y -320.479,Z 1324.691,A 0.000,B 0.000,C 90.000,E1 124.326} C_DIS
LIN {X 0.095,Y -322.405,Z 1324.689,A 0.000,B 0.000,C 90.000,E1 123.992} C_DIS
LIN {X -0.040,Y -323.903,Z 1324.687,A 0.000,B 0.000,C 90.000,E1 123.706} C_DIS
LIN {X -0.132,Y -336.731,Z 1324.668,A 0.000,B 0.000,C 90.000,E1 120.256} C_DIS
LIN {X -0.038,Y -348.612,Z 1324.653,A 0.000,B 0.000,C 90.000,E1 117.462} C_DIS
LIN {X 0.100,Y -361.941,Z 1324.637,A 0.000,B 0.000,C 90.000,E1 114.719} C_DIS
LIN {X -0.129,Y -375.104,Z 1324.624,A 0.000,B 0.000,C 90.000,E1 112.386} C_DIS
LIN {X -0.120,Y -389.598,Z 1324.611,A 0.000,B 0.000,C 90.000,E1 110.066} C_DIS
LIN {X 0.140,Y -405.523,Z 1324.599,A 0.000,B 0.000,C 90.000,E1 107.764} C_DIS
LIN {X 0.170,Y -422.993,Z 1324.587,A 0.000,B 0.000,C 90.000,E1 105.552} C_DIS
LIN {X 0.120,Y -442.101,Z 1324.575,A 0.000,B 0.000,C 90.000,E1 103.411} C_DIS
LIN {X -0.047,Y -462.182,Z 1324.563,A 0.000,B 0.000,C 90.000,E1 101.422} C_DIS
LIN {X -0.007,Y -477.598,Z 1324.556,A 0.000,B 0.000,C 90.000,E1 100.018} C_DIS
LIN {X -0.009,Y -479.970,Z 1324.554,A 0.000,B 0.000,C 90.000,E1 99.792} C_DIS
LIN {X -0.032,Y -481.849,Z 1324.553,A 0.000,B 0.000,C 90.000,E1 99.557} C_DIS
LIN {X -0.057,Y -483.274,Z 1324.552,A 0.000,B 0.000,C 90.000,E1 99.321} C_DIS
LIN {X 0.113,Y -485.194,Z 1324.549,A 0.000,B 0.000,C 90.000,E1 98.803} C_DIS
LIN {X -0.187,Y -485.991,Z 1324.546,A 0.000,B 0.000,C 90.000,E1 98.341} C_DIS
LIN {X 0.074,Y -485.800,Z 1324.543,A 0.000,B 0.000,C 90.000,E1 97.814} C_DIS
LIN {X -0.210,Y -484.596,Z 1324.541,A 0.000,B 0.000,C 90.000,E1 97.352} C_DIS
LIN {X 0.098,Y -483.555,Z 1324.539,A 0.000,B 0.000,C 90.000,E1 97.068} C_DIS
LIN {X -0.014,Y -482.155,Z 1324.538,A 0.000,B 0.000,C 90.000,E1 96.834} C_DIS
LIN {X 0.072,Y -467.666,Z 1324.527,A 0.000,B 0.000,C 90.000,E1 94.821} C_DIS
LIN {X -0.159,Y -454.094,Z 1324.516,A 0.000,B 0.000,C 90.000,E1 92.808} C_DIS
LIN {X 0.151,Y -440.961,Z 1324.504,A 0.000,B 0.000,C 90.000,E1 90.688} C_DIS
LIN {X -0.156,Y -423.157,Z 1324.486,A 0.000,B 0.000,C 90.000,E1 87.535} C_DIS
LIN {X -0.201,Y -413.033,Z 1324.476,A 0.000,B 0.000,C 90.000,E1 85.641} C_DIS
LIN {X -0.012,Y -402.765,Z 1324.465,A 0.000,B 0.000,C 90.000,E1 83.685} C_DIS
LIN {X -0.009,Y -392.253,Z 1324.454,A 0.000,B 0.000,C 90.000,E1 81.724} C_DIS
LIN {X -0.145,Y -382.928,Z 1324.445,A 0.000,B 0.000,C 90.000,E1 80.038} C_DIS
LIN {X -0.008,Y -374.982,Z 1324.437,A 0.000,B 0.000,C 90.000,E1 78.578} C_DIS
LIN {X -0.011,Y -365.253,Z 1324.427,A 0.000,B 0.000,C 90.000,E1 76.825} C_DIS
LIN {X -0.076,Y -353.746,Z 1324.415,A 0.000,B 0.000,C 90.000,E1 74.755} C_DIS
LIN {X 0.134,Y -343.830,Z 1324.405,A 0.000,B 0.000,C 90.000,E1 72.906} C_DIS
LIN {X -0.073,Y -332.220,Z 1324.393,A 0.000,B 0.000,C 90.000,E1 70.786} C_DIS
LIN {X -0.145,Y -319.273,Z 1324.379,A 0.000,B 0.000,C 90.000,E1 68.284} C_DIS
LIN {X -0.054,Y -302.575,Z 1324.359,A 0.000,B 0.000,C 90.000,E1 64.717} C_DIS
LIN {X -0.087,Y -293.119,Z 1324.347,A 0.000,B 0.000,C 90.000,E1 62.410} C_DIS
LIN {X -0.026,Y -285.896,Z 1324.335,A 0.000,B 0.000,C 90.000,E1 60.383} C_DIS
LIN {X 0.023,Y -275.407,Z 1324.317,A 0.000,B 0.000,C 90.000,E1 56.962} C_DIS
LIN {X -0.025,Y -266.003,Z 1324.297,A 0.000,B 0.000,C 90.000,E1 53.497} C_DIS
LIN {X 0.111,Y -258.925,Z 1324.281,A 0.000,B 0.000,C 90.000,E1 50.642} C_DIS
LIN {X 0.061,Y -250.602,Z 1324.262,A 0.000,B 0.000,C 90.000,E1 47.067} C_DIS
LIN {X -0.102,Y -242.581,Z 1324.241,A 0.000,B 0.000,C 90.000,E1 43.461} C_DIS
LIN {X 0.037,Y -235.093,Z 1324.221,A 0.000,B 0.000,C 90.000,E1 39.725} C_DIS
LIN {X 0.046,Y -228.514,Z 1324.200,A 0.000,B 0.000,C 90.000,E1 35.964} C_DIS
LIN {X 0.016,Y -222.930,Z 1324.179,A 0.000,B 0.000,C 90.000,E1 32.163} C_DIS
LIN {X 0.030,Y -218.335,Z 1324.157,A 0.000,B 0.000,C 90.000,E1 28.309} C_DIS
LIN {X -0.126,Y -214.563,Z 1324.136,A 0.000,B 0.000,C 90.000,E1 24.463} C_DIS
LIN {X 0.107,Y -211.213,Z 1324.114,A 0.000,B 0.000,C 90.000,E1 20.482} C_DIS
LIN {X -0.005,Y -208.230,Z 1324.092,A 0.000,B 0.000,C 90.000,E1 16.567} C_DIS
LIN {X -0.069,Y -206.028,Z 1324.074,A 0.000,B 0.000,C 90.000,E1 13.411} C_DIS
LIN {X 0.089,Y -203.547,Z 1324.052,A 0.000,B 0.000,C 90.000,E1 9.378} C_DIS
LIN {X 0.002,Y -200.962,Z 1324.021,A 0.000,B 0.000,C 90.000,E1 3.784} C_DIS
LIN {X -0.093,Y -199.651,Z 1323.984,A 0.000,B 0.000,C 90.000,E1 357.135} C_DIS
LIN {X -0.077,Y -200.572,Z 1323.943,A 0.000,B 0.000,C 90.000,E1 349.859} C_DIS
LIN {X 0.066,Y -203.463,Z 1323.908,A 0.000,B 0.000,C 90.000,E1 343.378} C_DIS
LIN {X 0.017,Y -207.230,Z 1323.881,A 0.000,B 0.000,C 90.000,E1 338.592} C_DIS
LIN {X -0.130,Y -211.350,Z 1323.859,A 0.000,B 0.000,C 90.000,E1 334.665} C_DIS
LIN {X -0.070,Y -216.416,Z 1323.837,A 0.000,B 0.000,C 90.000,E1 330.717} C_DIS
LIN {X -0.088,Y -222.521,Z 1323.816,A 0.000,B 0.000,C 90.000,E1 326.834} C_DIS
LIN {X 0.026,Y -229.528,Z 1323.794,A 0.000,B 0.000,C 90.000,E1 322.970} C_DIS
LIN {X -0.016,Y -235.984,Z 1323.777,A 0.000,B 0.000,C 90.000,E1 319.952} C_DIS
LIN {X 0.022,Y -245.033,Z 1323.757,A 0.000,B 0.000,C 90.000,E1 316.215} C_DIS
LIN {X -0.034,Y -253.254,Z 1323.740,A 0.000,B 0.000,C 90.000,E1 313.299} C_DIS
LIN {X -0.051,Y -261.444,Z 1323.727,A 0.000,B 0.000,C 90.000,E1 310.782} C_DIS
LIN {X 0.084,Y -269.281,Z 1323.715,A 0.000,B 0.000,C 90.000,E1 308.624} C_DIS
LIN {X 0.042,Y -278.052,Z 1323.703,A 0.000,B 0.000,C 90.000,E1 306.537} C_DIS
LIN {X 0.001,Y -287.856,Z 1323.692,A 0.000,B 0.000,C 90.000,E1 304.485} C_DIS
LIN {X -0.024,Y -298.732,Z 1323.680,A 0.000,B 0.000,C 90.000,E1 302.467} C_DIS
LIN {X 0.052,Y -308.853,Z 1323.671,A 0.000,B 0.000,C 90.000,E1 300.797} C_DIS
LIN {X -0.129,Y -320.096,Z 1323.662,A 0.000,B 0.000,C 90.000,E1 299.205} C_DIS
LIN {X 0.102,Y -335.009,Z 1323.651,A 0.000,B 0.000,C 90.000,E1 297.257} C_DIS
LIN {X 0.083,Y -353.457,Z 1323.640,A 0.000,B 0.000,C 90.000,E1 295.103} C_DIS
LIN {X 0.118,Y -368.950,Z 1323.630,A 0.000,B 0.000,C 90.000,E1 293.334} C_DIS
LIN {X -0.051,Y -381.547,Z 1323.622,A 0.000,B 0.000,C 90.000,E1 291.897} C_DIS
LIN {X 0.143,Y -393.662,Z 1323.614,A 0.000,B 0.000,C 90.000,E1 290.429} C_DIS
LIN {X -0.159,Y -413.310,Z 1323.601,A 0.000,B 0.000,C 90.000,E1 288.236} C_DIS
LIN {X 0.153,Y -423.047,Z 1323.595,A 0.000,B 0.000,C 90.000,E1 287.094} C_DIS
LIN {X -0.100,Y -430.007,Z 1323.591,A 0.000,B 0.000,C 90.000,E1 286.315} C_DIS
LIN {X 0.114,Y -436.495,Z 1323.586,A 0.000,B 0.000,C 90.000,E1 285.481} C_DIS
LIN {X -0.142,Y -442.363,Z 1323.582,A 0.000,B 0.000,C 90.000,E1 284.717} C_DIS
LIN {X 0.191,Y -447.532,Z 1323.577,A 0.000,B 0.000,C 90.000,E1 283.883} C_DIS
LIN {X 0.033,Y -452.012,Z 1323.573,A 0.000,B 0.000,C 90.000,E1 283.119} C_DIS
LIN {X -0.092,Y -455.802,Z 1323.569,A 0.000,B 0.000,C 90.000,E1 282.355} C_DIS
LIN {X -0.006,Y -457.974,Z 1323.566,A 0.000,B 0.000,C 90.000,E1 281.827} C_DIS
LIN {X 0.093,Y -459.791,Z 1323.563,A 0.000,B 0.000,C 90.000,E1 281.299} C_DIS
LIN {X 0.111,Y -461.242,Z 1323.560,A 0.000,B 0.000,C 90.000,E1 280.782} C_DIS
LIN {X 0.228,Y -462.316,Z 1323.557,A 0.000,B 0.000,C 90.000,E1 280.254} C_DIS
LIN {X -0.185,Y -462.998,Z 1323.554,A 0.000,B 0.000,C 90.000,E1 279.792} C_DIS
LIN {X -0.057,Y -463.228,Z 1323.551,A 0.000,B 0.000,C 90.000,E1 279.265} C_DIS
LIN {X 0.000,Y -463.041,Z 1323.549,A 0.000,B 0.000,C 90.000,E1 278.746} C_DIS
LIN {X 0.127,Y -462.434,Z 1323.546,A 0.000,B 0.000,C 90.000,E1 278.219} C_DIS
LIN {X 0.186,Y -461.274,Z 1323.543,A 0.000,B 0.000,C 90.000,E1 277.701} C_DIS
LIN {X -0.214,Y -459.640,Z 1323.540,A 0.000,B 0.000,C 90.000,E1 277.239} C_DIS
LIN {X -0.163,Y -457.501,Z 1323.537,A 0.000,B 0.000,C 90.000,E1 276.720} C_DIS
LIN {X -0.120,Y -454.852,Z 1323.534,A 0.000,B 0.000,C 90.000,E1 276.201} C_DIS
LIN {X -0.097,Y -451.584,Z 1323.531,A 0.000,B 0.000,C 90.000,E1 275.682} C_DIS
LIN {X -0.093,Y -447.674,Z 1323.529,A 0.000,B 0.000,C 90.000,E1 275.163} C_DIS
LIN {X -0.111,Y -442.931,Z 1323.526,A 0.000,B 0.000,C 90.000,E1 274.645} C_DIS
LIN {X -0.153,Y -437.252,Z 1323.523,A 0.000,B 0.000,C 90.000,E1 274.131} C_DIS
LIN {X -0.172,Y -431.263,Z 1323.520,A 0.000,B 0.000,C 90.000,E1 273.669} C_DIS
LIN {X 0.158,Y -424.927,Z 1323.518,A 0.000,B 0.000,C 90.000,E1 273.212} C_DIS
LIN {X 0.057,Y -418.285,Z 1323.516,A 0.000,B 0.000,C 90.000,E1 272.865} C_DIS
LIN {X -0.142,Y -411.508,Z 1323.514,A 0.000,B 0.000,C 90.000,E1 272.579} C_DIS
LIN {X -0.039,Y -404.505,Z 1323.513,A 0.000,B 0.000,C 90.000,E1 272.293} C_DIS
LIN {X -0.035,Y -397.516,Z 1323.511,A 0.000,B 0.000,C 90.000,E1 272.064} C_DIS
LIN {X 0.097,Y -386.360,Z 1323.510,A 0.000,B 0.000,C 90.000,E1 271.776} C_DIS
LIN {X -0.087,Y -378.662,Z 1323.509,A 0.000,B 0.000,C 90.000,E1 271.661} C_DIS
LIN {X -0.095,Y -369.553,Z 1323.509,A 0.000,B 0.000,C 90.000,E1 271.547} C_DIS
LIN {X 0.083,Y -355.926,Z 1323.508,A 0.000,B 0.000,C 90.000,E1 271.432} C_DIS
LIN {X -0.028,Y -349.272,Z 1323.508,A 0.000,B 0.000,C 90.000,E1 271.432} C_DIS
LIN {X -0.043,Y -181.368,Z 1323.508,A 0.000,B 0.000,C 90.000,E1 271.432} C_DIS
LIN {X -0.001,Y -181.575,Z 1323.502,A 0.000,B 0.000,C 90.000,E1 270.401} C_DIS
LIN {X 0.005,Y -180.893,Z 1323.473,A 0.000,B 0.000,C 90.000,E1 265.179} C_DIS
LIN {X 0.082,Y -179.518,Z 1323.454,A 0.000,B 0.000,C 90.000,E1 261.781} C_DIS
LIN {X 0.067,Y -179.021,Z 1323.445,A 0.000,B 0.000,C 90.000,E1 260.095} C_DIS
LIN {X -0.048,Y -178.656,Z 1323.440,A 0.000,B 0.000,C 90.000,E1 259.285} C_DIS
LIN {X 0.058,Y -175.706,Z 1323.412,A 0.000,B 0.000,C 90.000,E1 254.157} C_DIS
LIN {X 0.069,Y -172.422,Z 1323.388,A 0.000,B 0.000,C 90.000,E1 249.880} C_DIS
LIN {X 0.085,Y -171.244,Z 1323.379,A 0.000,B 0.000,C 90.000,E1 248.156} C_DIS
LIN {X -0.090,Y -167.520,Z 1323.355,A 0.000,B 0.000,C 90.000,E1 243.896} C_DIS
LIN {X -0.007,Y -166.915,Z 1323.350,A 0.000,B 0.000,C 90.000,E1 242.999} C_DIS
LIN {X 0.044,Y -162.223,Z 1323.321,A 0.000,B 0.000,C 90.000,E1 237.740} C_DIS
LIN {X -0.036,Y -160.806,Z 1323.311,A 0.000,B 0.000,C 90.000,E1 236.008} C_DIS
LIN {X -0.057,Y -157.592,Z 1323.291,A 0.000,B 0.000,C 90.000,E1 232.477} C_DIS
LIN {X 0.001,Y -155.626,Z 1323.277,A 0.000,B 0.000,C 90.000,E1 229.784} C_DIS
LIN {X -0.064,Y -151.902,Z 1323.252,A 0.000,B 0.000,C 90.000,E1 225.324} C_DIS
LIN {X -0.048,Y -150.133,Z 1323.237,A 0.000,B 0.000,C 90.000,E1 222.609} C_DIS
LIN {X 0.079,Y -146.921,Z 1323.211,A 0.000,B 0.000,C 90.000,E1 218.016} C_DIS
LIN {X -0.020,Y -145.508,Z 1323.196,A 0.000,B 0.000,C 90.000,E1 215.311} C_DIS
LIN {X -0.025,Y -142.911,Z 1323.171,A 0.000,B 0.000,C 90.000,E1 210.718} C_DIS
LIN {X 0.028,Y -141.533,Z 1323.150,A 0.000,B 0.000,C 90.000,E1 207.001} C_DIS
LIN {X 0.071,Y -139.400,Z 1323.114,A 0.000,B 0.000,C 90.000,E1 200.482} C_DIS
LIN {X -0.010,Y -139.113,Z 1323.104,A 0.000,B 0.000,C 90.000,E1 198.652} C_DIS
LIN {X -0.023,Y -138.352,Z 1323.057,A 0.000,B 0.000,C 90.000,E1 190.254} C_DIS
LIN {X -0.033,Y -139.506,Z 1323.005,A 0.000,B 0.000,C 90.000,E1 180.917} C_DIS
LIN {X 0.048,Y -141.144,Z 1322.974,A 0.000,B 0.000,C 90.000,E1 175.298} C_DIS
LIN {X 0.001,Y -142.524,Z 1322.958,A 0.000,B 0.000,C 90.000,E1 172.534} C_DIS
LIN {X -0.054,Y -144.789,Z 1322.933,A 0.000,B 0.000,C 90.000,E1 167.937} C_DIS
LIN {X 0.077,Y -147.406,Z 1322.912,A 0.000,B 0.000,C 90.000,E1 164.212} C_DIS
LIN {X -0.035,Y -149.981,Z 1322.892,A 0.000,B 0.000,C 90.000,E1 160.604} C_DIS
LIN {X -0.027,Y -153.306,Z 1322.872,A 0.000,B 0.000,C 90.000,E1 156.975} C_DIS
LIN {X -0.039,Y -155.008,Z 1322.862,A 0.000,B 0.000,C 90.000,E1 155.177} C_DIS
LIN {X 0.049,Y -158.652,Z 1322.842,A 0.000,B 0.000,C 90.000,E1 151.563} C_DIS
LIN {X -0.007,Y -161.928,Z 1322.827,A 0.000,B 0.000,C 90.000,E1 148.918} C_DIS
LIN {X 0.017,Y -166.118,Z 1322.808,A 0.000,B 0.000,C 90.000,E1 145.388} C_DIS
LIN {X 0.014,Y -171.128,Z 1322.788,A 0.000,B 0.000,C 90.000,E1 141.904} C_DIS
LIN {X -0.067,Y -176.006,Z 1322.769,A 0.000,B 0.000,C 90.000,E1 138.485} C_DIS
LIN {X 0.046,Y -180.255,Z 1322.755,A 0.000,B 0.000,C 90.000,E1 135.891} C_DIS
LIN {X 0.019,Y -185.669,Z 1322.736,A 0.000,B 0.000,C 90.000,E1 132.528} C_DIS
LIN {X 0.072,Y -190.270,Z 1322.722,A 0.000,B 0.000,C 90.000,E1 130.011} C_DIS
LIN {X -0.038,Y -197.598,Z 1322.700,A 0.000,B 0.000,C 90.000,E1 125.931} C_DIS
LIN {X -0.045,Y -199.251,Z 1322.695,A 0.000,B 0.000,C 90.000,E1 125.105} C_DIS
LIN {X -0.105,Y -308.723,Z 1322.695,A 0.000,B 0.000,C 90.000,E1 125.105} C_DIS
LIN {X 0.080,Y -311.266,Z 1322.695,A 0.000,B 0.000,C 90.000,E1 125.025} C_DIS
LIN {X 0.191,Y -315.131,Z 1322.694,A 0.000,B 0.000,C 90.000,E1 124.818} C_DIS
LIN {X -0.140,Y -317.437,Z 1322.693,A 0.000,B 0.000,C 90.000,E1 124.692} C_DIS
LIN {X 0.082,Y -320.614,Z 1322.691,A 0.000,B 0.000,C 90.000,E1 124.278} C_DIS
LIN {X -0.077,Y -322.534,Z 1322.689,A 0.000,B 0.000,C 90.000,E1 123.992} C_DIS
LIN {X 0.032,Y -324.025,Z 1322.687,A 0.000,B 0.000,C 90.000,E1 123.658} C_DIS
LIN {X 0.089,Y -338.102,Z 1322.666,A 0.000,B 0.000,C 90.000,E1 119.873} C_DIS
LIN {X -0.070,Y -350.151,Z 1322.651,A 0.000,B 0.000,C 90.000,E1 117.129} C_DIS
LIN {X 0.100,Y -363.672,Z 1322.636,A 0.000,B 0.000,C 90.000,E1 114.387} C_DIS
LIN {X 0.107,Y -377.014,Z 1322.622,A 0.000,B 0.000,C 90.000,E1 112.025} C_DIS
LIN {X -0.188,Y -391.701,Z 1322.610,A 0.000,B 0.000,C 90.000,E1 109.758} C_DIS
LIN {X 0.117,Y -407.834,Z 1322.597,A 0.000,B 0.000,C 90.000,E1 107.457} C_DIS
LIN {X 0.198,Y -425.528,Z 1322.585,A 0.000,B 0.000,C 90.000,E1 105.245} C_DIS
LIN {X 0.124,Y -444.847,Z 1322.573,A 0.000,B 0.000,C 90.000,E1 103.119} C_DIS
LIN {X 0.151,Y -465.005,Z 1322.562,A 0.000,B 0.000,C 90.000,E1 101.130} C_DIS
LIN {X 0.249,Y -477.863,Z 1322.556,A 0.000,B 0.000,C 90.000,E1 99.962} C_DIS
LIN {X -0.140,Y -480.144,Z 1322.554,A 0.000,B 0.000,C 90.000,E1 99.782} C_DIS
LIN {X 0.183,Y -481.984,Z 1322.553,A 0.000,B 0.000,C 90.000,E1 99.500} C_DIS
LIN {X 0.113,Y -483.374,Z 1322.552,A 0.000,B 0.000,C 90.000,E1 99.265} C_DIS
LIN {X -0.195,Y -485.183,Z 1322.549,A 0.000,B 0.000,C 90.000,E1 98.803} C_DIS
LIN {X 0.057,Y -485.889,Z 1322.546,A 0.000,B 0.000,C 90.000,E1 98.276} C_DIS
LIN {X 0.248,Y -485.612,Z 1322.543,A 0.000,B 0.000,C 90.000,E1 97.757} C_DIS
LIN {X -0.038,Y -484.310,Z 1322.541,A 0.000,B 0.000,C 90.000,E1 97.296} C_DIS
LIN {X -0.210,Y -483.211,Z 1322.539,A 0.000,B 0.000,C 90.000,E1 97.068} C_DIS
LIN {X 0.157,Y -481.738,Z 1322.538,A 0.000,B 0.000,C 90.000,E1 96.777} C_DIS
LIN {X -0.040,Y -468.924,Z 1322.528,A 0.000,B 0.000,C 90.000,E1 95.049} C_DIS
LIN {X 0.211,Y -455.305,Z 1322.517,A 0.000,B 0.000,C 90.000,E1 92.980} C_DIS
LIN {X 0.094,Y -442.055,Z 1322.505,A 0.000,B 0.000,C 90.000,E1 90.917} C_DIS
LIN {X -0.047,Y -422.720,Z 1322.486,A 0.000,B 0.000,C 90.000,E1 87.478} C_DIS
LIN {X -0.104,Y -412.584,Z 1322.475,A 0.000,B 0.000,C 90.000,E1 85.584} C_DIS
LIN {X 0.071,Y -402.331,Z 1322.465,A 0.000,B 0.000,C 90.000,E1 83.628} C_DIS
LIN {X 0.117,Y -391.816,Z 1322.454,A 0.000,B 0.000,C 90.000,E1 81.659} C_DIS
LIN {X -0.086,Y -382.505,Z 1322.444,A 0.000,B 0.000,C 90.000,E1 79.982} C_DIS
LIN {X 0.050,Y -372.942,Z 1322.435,A 0.000,B 0.000,C 90.000,E1 78.229} C_DIS
LIN {X 0.089,Y -363.181,Z 1322.425,A 0.000,B 0.000,C 90.000,E1 76.464} C_DIS
LIN {X -0.011,Y -351.664,Z 1322.413,A 0.000,B 0.000,C 90.000,E1 74.393} C_DIS
LIN {X 0.161,Y -341.726,Z 1322.403,A 0.000,B 0.000,C 90.000,E1 72.543} C_DIS
LIN {X -0.114,Y -328.483,Z 1322.389,A 0.000,B 0.000,C 90.000,E1 70.115} C_DIS
LIN {X 0.135,Y -315.693,Z 1322.375,A 0.000,B 0.000,C 90.000,E1 67.539} C_DIS
LIN {X -0.065,Y -300.796,Z 1322.357,A 0.000,B 0.000,C 90.000,E1 64.332} C_DIS
LIN {X -0.135,Y -292.792,Z 1322.346,A 0.000,B 0.000,C 90.000,E1 62.359} C_DIS
LIN {X -0.083,Y -285.615,Z 1322.335,A 0.000,B 0.000,C 90.000,E1 60.333} C_DIS
LIN {X -0.050,Y -275.169,Z 1322.316,A 0.000,B 0.000,C 90.000,E1 56.914} C_DIS
LIN {X 0.048,Y -265.797,Z 1322.297,A 0.000,B 0.000,C 90.000,E1 53.417} C_DIS
LIN {X 0.015,Y -258.753,Z 1322.281,A 0.000,B 0.000,C 90.000,E1 50.598} C_DIS
LIN {X -0.048,Y -250.434,Z 1322.261,A 0.000,B 0.000,C 90.000,E1 47.025} C_DIS
LIN {X -0.047,Y -242.422,Z 1322.241,A 0.000,B 0.000,C 90.000,E1 43.380} C_DIS
LIN {X 0.085,Y -234.941,Z 1322.220,A 0.000,B 0.000,C 90.000,E1 39.644} C_DIS
LIN {X 0.085,Y -228.380,Z 1322.199,A 0.000,B 0.000,C 90.000,E1 35.884} C_DIS
LIN {X 0.047,Y -222.797,Z 1322.178,A 0.000,B 0.000,C 90.000,E1 32.084} C_DIS
LIN {X 0.050,Y -218.206,Z 1322.157,A 0.000,B 0.000,C 90.000,E1 28.231} C_DIS
LIN {X 0.079,Y -214.419,Z 1322.135,A 0.000,B 0.000,C 90.000,E1 24.335} C_DIS
LIN {X 0.031,Y -211.039,Z 1322.114,A 0.000,B 0.000,C 90.000,E1 20.429} C_DIS
LIN {X -0.023,Y -208.035,Z 1322.092,A 0.000,B 0.000,C 90.000,E1 16.496} C_DIS
LIN {X -0.062,Y -205.284,Z 1322.070,A 0.000,B 0.000,C 90.000,E1 12.535} C_DIS
LIN {X 0.072,Y -202.474,Z 1322.043,A 0.000,B 0.000,C 90.000,E1 7.701} C_DIS
LIN {X 0.081,Y -200.088,Z 1322.007,A 0.000,B 0.000,C 90.000,E1 1.260} C_DIS
LIN {X 0.059,Y -199.537,Z 1321.970,A 0.000,B 0.000,C 90.000,E1 354.666} C_DIS
LIN {X -0.030,Y -201.054,Z 1321.935,A 0.000,B 0.000,C 90.000,E1 348.229} C_DIS
LIN {X -0.027,Y -204.007,Z 1321.903,A 0.000,B 0.000,C 90.000,E1 342.598} C_DIS
LIN {X 0.011,Y -208.028,Z 1321.877,A 0.000,B 0.000,C 90.000,E1 337.794} C_DIS
LIN {X -0.027,Y -212.334,Z 1321.855,A 0.000,B 0.000,C 90.000,E1 333.845} C_DIS
LIN {X -0.022,Y -217.654,Z 1321.833,A 0.000,B 0.000,C 90.000,E1 329.921} C_DIS
LIN {X 0.120,Y -223.950,Z 1321.811,A 0.000,B 0.000,C 90.000,E1 326.008} C_DIS
LIN {X 0.098,Y -231.165,Z 1321.790,A 0.000,B 0.000,C 90.000,E1 322.190} C_DIS
LIN {X 0.008,Y -239.561,Z 1321.769,A 0.000,B 0.000,C 90.000,E1 318.447} C_DIS
LIN {X -0.021,Y -248.055,Z 1321.751,A 0.000,B 0.000,C 90.000,E1 315.121} C_DIS
LIN {X 0.039,Y -257.872,Z 1321.732,A 0.000,B 0.000,C 90.000,E1 311.838} C_DIS
LIN {X -0.039,Y -266.647,Z 1321.719,A 0.000,B 0.000,C 90.000,E1 309.358} C_DIS
LIN {X 0.029,Y -275.106,Z 1321.707,A 0.000,B 0.000,C 90.000,E1 307.237} C_DIS
LIN {X -0.025,Y -282.917,Z 1321.697,A 0.000,B 0.000,C 90.000,E1 305.518} C_DIS
LIN {X -0.148,Y -293.229,Z 1321.686,A 0.000,B 0.000,C 90.000,E1 303.499} C_DIS
LIN {X 0.001,Y -302.727,Z 1321.677,A 0.000,B 0.000,C 90.000,E1 301.799} C_DIS
LIN {X 0.147,Y -313.289,Z 1321.667,A 0.000,B 0.000,C 90.000,E1 300.129} C_DIS
LIN {X -0.119,Y -324.992,Z 1321.659,A 0.000,B 0.000,C 90.000,E1 298.565} C_DIS
LIN {X 0.111,Y -348.096,Z 1321.643,A 0.000,B 0.000,C 90.000,E1 295.720} C_DIS
LIN {X 0.178,Y -361.205,Z 1321.635,A 0.000,B 0.000,C 90.000,E1 294.207} C_DIS
LIN {X -0.029,Y -371.415,Z 1321.628,A 0.000,B 0.000,C 90.000,E1 293.078} C_DIS
LIN {X 0.163,Y -383.914,Z 1321.620,A 0.000,B 0.000,C 90.000,E1 291.589} C_DIS
LIN {X -0.122,Y -400.859,Z 1321.609,A 0.000,B 0.000,C 90.000,E1 289.631} C_DIS
LIN {X 0.058,Y -415.674,Z 1321.600,A 0.000,B 0.000,C 90.000,E1 287.946} C_DIS
LIN {X -0.250,Y -427.624,Z 1321.592,A 0.000,B 0.000,C 90.000,E1 286.622} C_DIS
LIN {X -0.051,Y -434.291,Z 1321.588,A 0.000,B 0.000,C 90.000,E1 285.788} C_DIS
LIN {X 0.208,Y -440.400,Z 1321.583,A 0.000,B 0.000,C 90.000,E1 284.954} C_DIS
LIN {X -0.010,Y -445.763,Z 1321.579,A 0.000,B 0.000,C 90.000,E1 284.189} C_DIS
LIN {X -0.081,Y -450.478,Z 1321.574,A 0.000,B 0.000,C 90.000,E1 283.411} C_DIS
LIN {X 0.227,Y -454.506,Z 1321.570,A 0.000,B 0.000,C 90.000,E1 282.591} C_DIS
LIN {X 0.127,Y -457.911,Z 1321.566,A 0.000,B 0.000,C 90.000,E1 281.827} C_DIS
LIN {X 0.225,Y -459.780,Z 1321.563,A 0.000,B 0.000,C 90.000,E1 281.299} C_DIS
LIN {X -0.209,Y -461.293,Z 1321.560,A 0.000,B 0.000,C 90.000,E1 280.838} C_DIS
LIN {X -0.094,Y -462.418,Z 1321.557,A 0.000,B 0.000,C 90.000,E1 280.310} C_DIS
LIN {X -0.051,Y -463.090,Z 1321.554,A 0.000,B 0.000,C 90.000,E1 279.792} C_DIS
LIN {X 0.077,Y -463.381,Z 1321.552,A 0.000,B 0.000,C 90.000,E1 279.265} C_DIS
LIN {X 0.135,Y -463.243,Z 1321.549,A 0.000,B 0.000,C 90.000,E1 278.746} C_DIS
LIN {X -0.195,Y -462.656,Z 1321.546,A 0.000,B 0.000,C 90.000,E1 278.276} C_DIS
LIN {X -0.134,Y -461.554,Z 1321.543,A 0.000,B 0.000,C 90.000,E1 277.757} C_DIS
LIN {X -0.077,Y -459.967,Z 1321.540,A 0.000,B 0.000,C 90.000,E1 277.239} C_DIS
LIN {X -0.024,Y -457.887,Z 1321.537,A 0.000,B 0.000,C 90.000,E1 276.720} C_DIS
LIN {X 0.019,Y -455.312,Z 1321.534,A 0.000,B 0.000,C 90.000,E1 276.201} C_DIS
LIN {X 0.043,Y -452.113,Z 1321.532,A 0.000,B 0.000,C 90.000,E1 275.682} C_DIS
LIN {X 0.049,Y -448.313,Z 1321.529,A 0.000,B 0.000,C 90.000,E1 275.163} C_DIS
LIN {X 0.033,Y -443.707,Z 1321.526,A 0.000,B 0.000,C 90.000,E1 274.645} C_DIS
LIN {X -0.039,Y -438.138,Z 1321.523,A 0.000,B 0.000,C 90.000,E1 274.131} C_DIS
LIN {X -0.151,Y -432.066,Z 1321.520,A 0.000,B 0.000,C 90.000,E1 273.669} C_DIS
LIN {X 0.117,Y -425.724,Z 1321.518,A 0.000,B 0.000,C 90.000,E1 273.212} C_DIS
LIN {X -0.025,Y -419.116,Z 1321.516,A 0.000,B 0.000,C 90.000,E1 272.865} C_DIS
LIN {X 0.160,Y -412.259,Z 1321.514,A 0.000,B 0.000,C 90.000,E1 272.522} C_DIS
LIN {X -0.164,Y -405.292,Z 1321.513,A 0.000,B 0.000,C 90.000,E1 272.293} C_DIS
LIN {X 0.190,Y -397.975,Z 1321.511,A 0.000,B 0.000,C 90.000,E1 272.007} C_DIS
LIN {X 0.059,Y -390.682,Z 1321.510,A 0.000,B 0.000,C 90.000,E1 271.835} C_DIS
LIN {X 0.156,Y -383.123,Z 1321.509,A 0.000,B 0.000,C 90.000,E1 271.661} C_DIS
LIN {X 0.042,Y -374.534,Z 1321.509,A 0.000,B 0.000,C 90.000,E1 271.547} C_DIS
LIN {X 0.026,Y -360.012,Z 1321.508,A 0.000,B 0.000,C 90.000,E1 271.432} C_DIS
LIN {X -0.140,Y -352.916,Z 1321.508,A 0.000,B 0.000,C 90.000,E1 271.432} C_DIS
LIN {X 0.081,Y -181.370,Z 1321.508,A 0.000,B 0.000,C 90.000,E1 271.375} C_DIS
LIN {X -0.085,Y -181.578,Z 1321.502,A 0.000,B 0.000,C 90.000,E1 270.401} C_DIS
LIN {X -0.080,Y -180.890,Z 1321.473,A 0.000,B 0.000,C 90.000,E1 265.179} C_DIS
LIN {X -0.017,Y -179.014,Z 1321.445,A 0.000,B 0.000,C 90.000,E1 260.095} C_DIS
LIN {X 0.077,Y -178.637,Z 1321.440,A 0.000,B 0.000,C 90.000,E1 259.218} C_DIS
LIN {X -0.024,Y -175.689,Z 1321.412,A 0.000,B 0.000,C 90.000,E1 254.157} C_DIS
LIN {X -0.013,Y -172.405,Z 1321.388,A 0.000,B 0.000,C 90.000,E1 249.880} C_DIS
LIN {X 0.004,Y -171.217,Z 1321.379,A 0.000,B 0.000,C 90.000,E1 248.156} C_DIS
LIN {X -0.020,Y -167.500,Z 1321.355,A 0.000,B 0.000,C 90.000,E1 243.845} C_DIS
LIN {X -0.088,Y -166.896,Z 1321.350,A 0.000,B 0.000,C 90.000,E1 242.999} C_DIS
LIN {X -0.035,Y -162.203,Z 1321.321,A 0.000,B 0.000,C 90.000,E1 237.740} C_DIS
LIN {X 0.019,Y -160.777,Z 1321.311,A 0.000,B 0.000,C 90.000,E1 235.960} C_DIS
LIN {X -0.010,Y -157.570,Z 1321.291,A 0.000,B 0.000,C 90.000,E1 232.431} C_DIS
LIN {X 0.024,Y -155.601,Z 1321.276,A 0.000,B 0.000,C 90.000,E1 229.747} C_DIS
LIN {X 0.075,Y -151.882,Z 1321.251,A 0.000,B 0.000,C 90.000,E1 225.243} C_DIS
LIN {X 0.088,Y -150.108,Z 1321.236,A 0.000,B 0.000,C 90.000,E1 222.528} C_DIS
LIN {X 0.005,Y -146.904,Z 1321.211,A 0.000,B 0.000,C 90.000,E1 218.016} C_DIS
LIN {X 0.025,Y -145.492,Z 1321.196,A 0.000,B 0.000,C 90.000,E1 215.264} C_DIS
LIN {X 0.025,Y -142.898,Z 1321.170,A 0.000,B 0.000,C 90.000,E1 210.669} C_DIS
LIN {X -0.044,Y -141.518,Z 1321.150,A 0.000,B 0.000,C 90.000,E1 207.001} C_DIS
LIN {X -0.001,Y -139.394,Z 1321.114,A 0.000,B 0.000,C 90.000,E1 200.482} C_DIS
LIN {X 0.049,Y -139.105,Z 1321.103,A 0.000,B 0.000,C 90.000,E1 198.598} C_DIS
LIN {X 0.042,Y -138.353,Z 1321.057,A 0.000,B 0.000,C 90.000,E1 190.197} C_DIS
LIN {X 0.035,Y -139.511,Z 1321.005,A 0.000,B 0.000,C 90.000,E1 180.859} C_DIS
LIN {X -0.024,Y -141.157,Z 1320.974,A 0.000,B 0.000,C 90.000,E1 175.298} C_DIS
LIN {X -0.053,Y -142.537,Z 1320.958,A 0.000,B 0.000,C 90.000,E1 172.527} C_DIS
LIN {X 0.014,Y -144.807,Z 1320.933,A 0.000,B 0.000,C 90.000,E1 167.881} C_DIS
LIN {X 0.002,Y -147.427,Z 1320.912,A 0.000,B 0.000,C 90.000,E1 164.212} C_DIS
LIN {X 0.031,Y -150.005,Z 1320.892,A 0.000,B 0.000,C 90.000,E1 160.550} C_DIS
LIN {X 0.038,Y -153.336,Z 1320.872,A 0.000,B 0.000,C 90.000,E1 156.922} C_DIS
LIN {X 0.019,Y -155.871,Z 1320.857,A 0.000,B 0.000,C 90.000,E1 154.229} C_DIS
LIN {X -0.014,Y -159.724,Z 1320.837,A 0.000,B 0.000,C 90.000,E1 150.667} C_DIS
LIN {X 0.053,Y -161.963,Z 1320.827,A 0.000,B 0.000,C 90.000,E1 148.869} C_DIS
LIN {X -0.063,Y -166.155,Z 1320.808,A 0.000,B 0.000,C 90.000,E1 145.388} C_DIS
LIN {X -0.068,Y -171.168,Z 1320.788,A 0.000,B 0.000,C 90.000,E1 141.904} C_DIS
LIN {X -0.033,Y -176.048,Z 1320.769,A 0.000,B 0.000,C 90.000,E1 138.447} C_DIS
LIN {X -0.038,Y -180.303,Z 1320.755,A 0.000,B 0.000,C 90.000,E1 135.891} C_DIS
LIN {X -0.067,Y -185.715,Z 1320.736,A 0.000,B 0.000,C 90.000,E1 132.528} C_DIS
LIN {X -0.015,Y -190.322,Z 1320.722,A 0.000,B 0.000,C 90.000,E1 130.011} C_DIS
LIN {X 0.032,Y -197.648,Z 1320.699,A 0.000,B 0.000,C 90.000,E1 125.884} C_DIS
LIN {X -0.063,Y -199.261,Z 1320.695,A 0.000,B 0.000,C 90.000,E1 125.105} C_DIS
LIN {X -0.138,Y -308.588,Z 1320.695,A 0.000,B 0.000,C 90.000,E1 125.105} C_DIS
LIN {X 0.053,Y -312.538,Z 1320.694,A 0.000,B 0.000,C 90.000,E1 124.978} C_DIS
LIN {X -0.017,Y -315.571,Z 1320.693,A 0.000,B 0.000,C 90.000,E1 124.818} C_DIS
LIN {X -0.092,Y -319.227,Z 1320.692,A 0.000,B 0.000,C 90.000,E1 124.485} C_DIS
LIN {X 0.104,Y -322.750,Z 1320.688,A 0.000,B 0.000,C 90.000,E1 123.913} C_DIS
LIN {X -0.086,Y -324.216,Z 1320.687,A 0.000,B 0.000,C 90.000,E1 123.627} C_DIS
LIN {X 0.103,Y -337.039,Z 1320.667,A 0.000,B 0.000,C 90.000,E1 120.129} C_DIS
LIN {X -0.089,Y -348.960,Z 1320.652,A 0.000,B 0.000,C 90.000,E1 117.385} C_DIS
LIN {X 0.045,Y -362.340,Z 1320.637,A 0.000,B 0.000,C 90.000,E1 114.643} C_DIS
LIN {X 0.020,Y -375.547,Z 1320.624,A 0.000,B 0.000,C 90.000,E1 112.280} C_DIS
LIN {X 0.192,Y -390.090,Z 1320.611,A 0.000,B 0.000,C 90.000,E1 109.939} C_DIS
LIN {X 0.084,Y -406.068,Z 1320.598,A 0.000,B 0.000,C 90.000,E1 107.692} C_DIS
LIN {X 0.115,Y -423.595,Z 1320.586,A 0.000,B 0.000,C 90.000,E1 105.481} C_DIS
LIN {X -0.034,Y -442.762,Z 1320.574,A 0.000,B 0.000,C 90.000,E1 103.355} C_DIS
LIN {X -0.157,Y -462.863,Z 1320.563,A 0.000,B 0.000,C 90.000,E1 101.366} C_DIS
LIN {X -0.084,Y -478.286,Z 1320.555,A 0.000,B 0.000,C 90.000,E1 99.962} C_DIS
LIN {X -0.010,Y -480.433,Z 1320.554,A 0.000,B 0.000,C 90.000,E1 99.726} C_DIS
LIN {X -0.014,Y -482.062,Z 1320.553,A 0.000,B 0.000,C 90.000,E1 99.500} C_DIS
LIN {X -0.133,Y -483.429,Z 1320.551,A 0.000,B 0.000,C 90.000,E1 99.265} C_DIS
LIN {X 0.224,Y -484.439,Z 1320.550,A 0.000,B 0.000,C 90.000,E1 98.973} C_DIS
LIN {X -0.075,Y -485.587,Z 1320.547,A 0.000,B 0.000,C 90.000,E1 98.511} C_DIS
LIN {X 0.113,Y -485.725,Z 1320.544,A 0.000,B 0.000,C 90.000,E1 97.992} C_DIS
LIN {X -0.172,Y -484.875,Z 1320.542,A 0.000,B 0.000,C 90.000,E1 97.530} C_DIS
LIN {X 0.085,Y -482.896,Z 1320.539,A 0.000,B 0.000,C 90.000,E1 97.004} C_DIS
LIN {X -0.089,Y -481.359,Z 1320.538,A 0.000,B 0.000,C 90.000,E1 96.777} C_DIS
LIN {X 0.187,Y -468.512,Z 1320.528,A 0.000,B 0.000,C 90.000,E1 94.992} C_DIS
LIN {X -0.032,Y -454.895,Z 1320.516,A 0.000,B 0.000,C 90.000,E1 92.980} C_DIS
LIN {X -0.151,Y -441.642,Z 1320.505,A 0.000,B 0.000,C 90.000,E1 90.917} C_DIS
LIN {X 0.121,Y -422.314,Z 1320.486,A 0.000,B 0.000,C 90.000,E1 87.421} C_DIS
LIN {X 0.055,Y -412.172,Z 1320.475,A 0.000,B 0.000,C 90.000,E1 85.527} C_DIS
LIN {X -0.187,Y -401.938,Z 1320.464,A 0.000,B 0.000,C 90.000,E1 83.628} C_DIS
LIN {X 0.184,Y -392.954,Z 1320.455,A 0.000,B 0.000,C 90.000,E1 81.894} C_DIS
LIN {X 0.061,Y -383.709,Z 1320.446,A 0.000,B 0.000,C 90.000,E1 80.208} C_DIS
LIN {X 0.148,Y -374.166,Z 1320.436,A 0.000,B 0.000,C 90.000,E1 78.465} C_DIS
LIN {X -0.149,Y -364.449,Z 1320.426,A 0.000,B 0.000,C 90.000,E1 76.756} C_DIS
LIN {X 0.128,Y -352.925,Z 1320.415,A 0.000,B 0.000,C 90.000,E1 74.629} C_DIS
LIN {X -0.006,Y -342.993,Z 1320.405,A 0.000,B 0.000,C 90.000,E1 72.834} C_DIS
LIN {X -0.037,Y -329.712,Z 1320.391,A 0.000,B 0.000,C 90.000,E1 70.369} C_DIS
LIN {X -0.060,Y -316.889,Z 1320.377,A 0.000,B 0.000,C 90.000,E1 67.847} C_DIS
LIN {X 0.059,Y -301.892,Z 1320.359,A 0.000,B 0.000,C 90.000,E1 64.588} C_DIS
LIN {X 0.006,Y -293.781,Z 1320.348,A 0.000,B 0.000,C 90.000,E1 62.615} C_DIS
LIN {X 0.074,Y -286.497,Z 1320.337,A 0.000,B 0.000,C 90.000,E1 60.589} C_DIS
LIN {X -0.015,Y -275.954,Z 1320.318,A 0.000,B 0.000,C 90.000,E1 57.199} C_DIS
LIN {X 0.101,Y -266.530,Z 1320.298,A 0.000,B 0.000,C 90.000,E1 53.703} C_DIS
LIN {X 0.086,Y -259.468,Z 1320.283,A 0.000,B 0.000,C 90.000,E1 50.884} C_DIS
LIN {X 0.048,Y -251.109,Z 1320.263,A 0.000,B 0.000,C 90.000,E1 47.310} C_DIS
LIN {X -0.099,Y -243.051,Z 1320.243,A 0.000,B 0.000,C 90.000,E1 43.704} C_DIS
LIN {X 0.103,Y -236.976,Z 1320.226,A 0.000,B 0.000,C 90.000,E1 40.701} C_DIS
LIN {X -0.059,Y -230.117,Z 1320.205,A 0.000,B 0.000,C 90.000,E1 36.996} C_DIS
LIN {X 0.078,Y -224.242,Z 1320.184,A 0.000,B 0.000,C 90.000,E1 33.166} C_DIS
LIN {X 0.045,Y -219.379,Z 1320.163,A 0.000,B 0.000,C 90.000,E1 29.333} C_DIS
LIN {X -0.036,Y -214.649,Z 1320.137,A 0.000,B 0.000,C 90.000,E1 24.695} C_DIS
LIN {X -0.082,Y -211.201,Z 1320.115,A 0.000,B 0.000,C 90.000,E1 20.791} C_DIS
LIN {X 0.070,Y -208.105,Z 1320.094,A 0.000,B 0.000,C 90.000,E1 16.804} C_DIS
LIN {X 0.086,Y -205.332,Z 1320.071,A 0.000,B 0.000,C 90.000,E1 12.827} C_DIS
LIN {X 0.046,Y -202.067,Z 1320.040,A 0.000,B 0.000,C 90.000,E1 7.239} C_DIS
LIN {X 0.000,Y -199.682,Z 1320.000,A 0.000,B 0.000,C 90.000,E1 360.000} C_DIS
LIN {X 0.044,Y -199.771,Z 1319.957,A 0.000,B 0.000,C 90.000,E1 352.243} C_DIS
LIN {X -0.036,Y -202.051,Z 1319.921,A 0.000,B 0.000,C 90.000,E1 345.811} C_DIS
LIN {X 0.064,Y -205.231,Z 1319.894,A 0.000,B 0.000,C 90.000,E1 340.967} C_DIS
LIN {X -0.087,Y -209.708,Z 1319.868,A 0.000,B 0.000,C 90.000,E1 336.230} C_DIS
LIN {X -0.078,Y -214.386,Z 1319.846,A 0.000,B 0.000,C 90.000,E1 332.281} C_DIS
LIN {X 0.107,Y -220.151,Z 1319.824,A 0.000,B 0.000,C 90.000,E1 328.329} C_DIS
LIN {X 0.074,Y -226.840,Z 1319.803,A 0.000,B 0.000,C 90.000,E1 324.482} C_DIS
LIN {X -0.091,Y -234.486,Z 1319.782,A 0.000,B 0.000,C 90.000,E1 320.723} C_DIS
LIN {X -0.105,Y -243.285,Z 1319.761,A 0.000,B 0.000,C 90.000,E1 316.986} C_DIS
LIN {X -0.027,Y -252.321,Z 1319.743,A 0.000,B 0.000,C 90.000,E1 313.662} C_DIS
LIN {X -0.084,Y -260.342,Z 1319.729,A 0.000,B 0.000,C 90.000,E1 311.148} C_DIS
LIN {X 0.097,Y -269.419,Z 1319.715,A 0.000,B 0.000,C 90.000,E1 308.624} C_DIS
LIN {X -0.068,Y -279.749,Z 1319.701,A 0.000,B 0.000,C 90.000,E1 306.217} C_DIS
LIN {X 0.128,Y -291.506,Z 1319.688,A 0.000,B 0.000,C 90.000,E1 303.785} C_DIS
LIN {X -0.001,Y -300.804,Z 1319.678,A 0.000,B 0.000,C 90.000,E1 302.133} C_DIS
LIN {X 0.119,Y -311.168,Z 1319.669,A 0.000,B 0.000,C 90.000,E1 300.463} C_DIS
LIN {X -0.032,Y -322.660,Z 1319.660,A 0.000,B 0.000,C 90.000,E1 298.871} C_DIS
LIN {X -0.055,Y -345.510,Z 1319.645,A 0.000,B 0.000,C 90.000,E1 296.052} C_DIS
LIN {X 0.125,Y -358.610,Z 1319.636,A 0.000,B 0.000,C 90.000,E1 294.515} C_DIS
LIN {X -0.162,Y -371.620,Z 1319.628,A 0.000,B 0.000,C 90.000,E1 293.078} C_DIS
LIN {X -0.101,Y -381.641,Z 1319.622,A 0.000,B 0.000,C 90.000,E1 291.897} C_DIS
LIN {X 0.095,Y -393.726,Z 1319.614,A 0.000,B 0.000,C 90.000,E1 290.429} C_DIS
LIN {X 0.158,Y -413.424,Z 1319.601,A 0.000,B 0.000,C 90.000,E1 288.181} C_DIS
LIN {X 0.076,Y -423.172,Z 1319.595,A 0.000,B 0.000,C 90.000,E1 287.094} C_DIS
LIN {X -0.178,Y -430.170,Z 1319.590,A 0.000,B 0.000,C 90.000,E1 286.315} C_DIS
LIN {X 0.037,Y -436.658,Z 1319.586,A 0.000,B 0.000,C 90.000,E1 285.481} C_DIS
LIN {X -0.219,Y -442.453,Z 1319.582,A 0.000,B 0.000,C 90.000,E1 284.717} C_DIS
LIN {X 0.113,Y -447.541,Z 1319.577,A 0.000,B 0.000,C 90.000,E1 283.883} C_DIS
LIN {X -0.045,Y -451.993,Z 1319.573,A 0.000,B 0.000,C 90.000,E1 283.119} C_DIS
LIN {X -0.169,Y -455.814,Z 1319.568,A 0.000,B 0.000,C 90.000,E1 282.355} C_DIS
LIN {X -0.084,Y -457.999,Z 1319.566,A 0.000,B 0.000,C 90.000,E1 281.827} C_DIS
LIN {X 0.015,Y -459.885,Z 1319.563,A 0.000,B 0.000,C 90.000,E1 281.299} C_DIS
LIN {X 0.033,Y -461.409,Z 1319.560,A 0.000,B 0.000,C 90.000,E1 280.782} C_DIS
LIN {X 0.150,Y -462.529,Z 1319.557,A 0.000,B 0.000,C 90.000,E1 280.254} C_DIS
LIN {X -0.184,Y -463.238,Z 1319.554,A 0.000,B 0.000,C 90.000,E1 279.782} C_DIS
LIN {X -0.133,Y -463.534,Z 1319.551,A 0.000,B 0.000,C 90.000,E1 279.265} C_DIS
LIN {X -0.075,Y -463.380,Z 1319.549,A 0.000,B 0.000,C 90.000,E1 278.746} C_DIS
LIN {X 0.055,Y -462.771,Z 1319.546,A 0.000,B 0.000,C 90.000,E1 278.219} C_DIS
LIN {X 0.116,Y -461.703,Z 1319.543,A 0.000,B 0.000,C 90.000,E1 277.701} C_DIS
LIN {X 0.174,Y -460.145,Z 1319.540,A 0.000,B 0.000,C 90.000,E1 277.182} C_DIS
LIN {X -0.228,Y -458.070,Z 1319.537,A 0.000,B 0.000,C 90.000,E1 276.720} C_DIS
LIN {X -0.182,Y -455.527,Z 1319.534,A 0.000,B 0.000,C 90.000,E1 276.201} C_DIS
LIN {X -0.156,Y -452.388,Z 1319.531,A 0.000,B 0.000,C 90.000,E1 275.682} C_DIS
LIN {X -0.148,Y -448.614,Z 1319.529,A 0.000,B 0.000,C 90.000,E1 275.163} C_DIS
LIN {X -0.160,Y -444.040,Z 1319.526,A 0.000,B 0.000,C 90.000,E1 274.645} C_DIS
LIN {X -0.228,Y -438.540,Z 1319.523,A 0.000,B 0.000,C 90.000,E1 274.131} C_DIS
LIN {X 0.076,Y -432.459,Z 1319.520,A 0.000,B 0.000,C 90.000,E1 273.612} C_DIS
LIN {X -0.087,Y -426.115,Z 1319.518,A 0.000,B 0.000,C 90.000,E1 273.212} C_DIS
LIN {X 0.195,Y -419.571,Z 1319.516,A 0.000,B 0.000,C 90.000,E1 272.808} C_DIS
LIN {X -0.050,Y -412.680,Z 1319.514,A 0.000,B 0.000,C 90.000,E1 272.522} C_DIS
LIN {X 0.035,Y -405.753,Z 1319.512,A 0.000,B 0.000,C 90.000,E1 272.236} C_DIS
LIN {X 0.008,Y -398.467,Z 1319.511,A 0.000,B 0.000,C 90.000,E1 272.007} C_DIS
LIN {X -0.114,Y -391.283,Z 1319.510,A 0.000,B 0.000,C 90.000,E1 271.835} C_DIS
LIN {X -0.038,Y -383.476,Z 1319.509,A 0.000,B 0.000,C 90.000,E1 271.661} C_DIS
LIN {X -0.127,Y -375.031,Z 1319.509,A 0.000,B 0.000,C 90.000,E1 271.547} C_DIS
LIN {X -0.132,Y -360.892,Z 1319.508,A 0.000,B 0.000,C 90.000,E1 271.432} C_DIS
LIN {X 0.006,Y -347.636,Z 1319.508,A 0.000,B 0.000,C 90.000,E1 271.375} C_DIS
LIN {X -0.025,Y -181.378,Z 1319.508,A 0.000,B 0.000,C 90.000,E1 271.375} C_DIS
LIN {X 0.019,Y -181.579,Z 1319.502,A 0.000,B 0.000,C 90.000,E1 270.344} C_DIS
LIN {X 0.023,Y -180.886,Z 1319.473,A 0.000,B 0.000,C 90.000,E1 265.122} C_DIS
LIN {X 0.082,Y -179.008,Z 1319.445,A 0.000,B 0.000,C 90.000,E1 260.038} C_DIS
LIN {X 0.001,Y -178.620,Z 1319.440,A 0.000,B 0.000,C 90.000,E1 259.218} C_DIS
LIN {X 0.068,Y -175.672,Z 1319.412,A 0.000,B 0.000,C 90.000,E1 254.102} C_DIS
LIN {X -0.088,Y -172.389,Z 1319.388,A 0.000,B 0.000,C 90.000,E1 249.880} C_DIS
LIN {X -0.072,Y -171.191,Z 1319.379,A 0.000,B 0.000,C 90.000,E1 248.156} C_DIS
LIN {X -0.021,Y -167.482,Z 1319.354,A 0.000,B 0.000,C 90.000,E1 243.819} C_DIS
LIN {X -0.012,Y -166.879,Z 1319.350,A 0.000,B 0.000,C 90.000,E1 242.948} C_DIS
LIN {X -0.021,Y -162.183,Z 1319.321,A 0.000,B 0.000,C 90.000,E1 237.709} C_DIS
LIN {X 0.037,Y -160.751,Z 1319.311,A 0.000,B 0.000,C 90.000,E1 235.928} C_DIS
LIN {X 0.015,Y -157.550,Z 1319.291,A 0.000,B 0.000,C 90.000,E1 232.396} C_DIS
LIN {X -0.047,Y -155.578,Z 1319.276,A 0.000,B 0.000,C 90.000,E1 229.747} C_DIS
LIN {X 0.005,Y -151.863,Z 1319.251,A 0.000,B 0.000,C 90.000,E1 225.243} C_DIS
LIN {X 0.019,Y -150.087,Z 1319.236,A 0.000,B 0.000,C 90.000,E1 222.528} C_DIS
LIN {X -0.064,Y -146.888,Z 1319.211,A 0.000,B 0.000,C 90.000,E1 218.016} C_DIS
LIN {X 0.041,Y -145.475,Z 1319.196,A 0.000,B 0.000,C 90.000,E1 215.231} C_DIS
LIN {X -0.042,Y -142.886,Z 1319.170,A 0.000,B 0.000,C 90.000,E1 210.669} C_DIS
LIN {X 0.015,Y -141.504,Z 1319.150,A 0.000,B 0.000,C 90.000,E1 206.950} C_DIS
LIN {X 0.063,Y -139.390,Z 1319.114,A 0.000,B 0.000,C 90.000,E1 200.429} C_DIS
LIN {X -0.016,Y -139.096,Z 1319.103,A 0.000,B 0.000,C 90.000,E1 198.598} C_DIS
LIN {X -0.024,Y -138.353,Z 1319.057,A 0.000,B 0.000,C 90.000,E1 190.197} C_DIS
LIN {X -0.031,Y -139.515,Z 1319.005,A 0.000,B 0.000,C 90.000,E1 180.859} C_DIS
LIN {X 0.049,Y -141.169,Z 1318.974,A 0.000,B 0.000,C 90.000,E1 175.241} C_DIS
LIN {X 0.021,Y -142.548,Z 1318.958,A 0.000,B 0.000,C 90.000,E1 172.470} C_DIS
LIN {X -0.054,Y -144.824,Z 1318.932,A 0.000,B 0.000,C 90.000,E1 167.881} C_DIS
LIN {X 0.075,Y -147.446,Z 1318.912,A 0.000,B 0.000,C 90.000,E1 164.157} C_DIS
LIN {X -0.039,Y -150.026,Z 1318.892,A 0.000,B 0.000,C 90.000,E1 160.550} C_DIS
LIN {X -0.032,Y -153.363,Z 1318.872,A 0.000,B 0.000,C 90.000,E1 156.922} C_DIS
LIN {X 0.016,Y -155.896,Z 1318.857,A 0.000,B 0.000,C 90.000,E1 154.204} C_DIS
LIN {X -0.087,Y -159.756,Z 1318.837,A 0.000,B 0.000,C 90.000,E1 150.667} C_DIS
LIN {X -0.020,Y -161.996,Z 1318.827,A 0.000,B 0.000,C 90.000,E1 148.869} C_DIS
LIN {X -0.001,Y -166.188,Z 1318.807,A 0.000,B 0.000,C 90.000,E1 145.341} C_DIS
LIN {X 0.097,Y -171.203,Z 1318.788,A 0.000,B 0.000,C 90.000,E1 141.823} C_DIS
LIN {X 0.022,Y -176.087,Z 1318.769,A 0.000,B 0.000,C 90.000,E1 138.405} C_DIS
LIN {X -0.117,Y -180.347,Z 1318.755,A 0.000,B 0.000,C 90.000,E1 135.891} C_DIS
LIN {X -0.009,Y -185.757,Z 1318.736,A 0.000,B 0.000,C 90.000,E1 132.486} C_DIS
LIN {X -0.095,Y -190.369,Z 1318.722,A 0.000,B 0.000,C 90.000,E1 130.011} C_DIS
LIN {X -0.050,Y -197.695,Z 1318.699,A 0.000,B 0.000,C 90.000,E1 125.884} C_DIS
LIN {X -0.080,Y -199.272,Z 1318.695,A 0.000,B 0.000,C 90.000,E1 125.105} C_DIS
LIN {X -0.171,Y -308.657,Z 1318.695,A 0.000,B 0.000,C 90.000,E1 125.105} C_DIS
LIN {X 0.165,Y -310.091,Z 1318.695,A 0.000,B 0.000,C 90.000,E1 125.025} C_DIS
LIN {X 0.062,Y -313.107,Z 1318.694,A 0.000,B 0.000,C 90.000,E1 124.945} C_DIS
LIN {X 0.062,Y -316.346,Z 1318.693,A 0.000,B 0.000,C 90.000,E1 124.739} C_DIS
LIN {X 0.037,Y -320.005,Z 1318.691,A 0.000,B 0.000,C 90.000,E1 124.358} C_DIS
LIN {X 0.012,Y -321.932,Z 1318.689,A 0.000,B 0.000,C 90.000,E1 124.072} C_DIS
LIN {X -0.013,Y -323.445,Z 1318.688,A 0.000,B 0.000,C 90.000,E1 123.785} C_DIS
LIN {X -0.109,Y -325.852,Z 1318.684,A 0.000,B 0.000,C 90.000,E1 123.166} C_DIS
LIN {X -0.112,Y -336.341,Z 1318.668,A 0.000,B 0.000,C 90.000,E1 120.335} C_DIS
LIN {X 0.139,Y -348.179,Z 1318.653,A 0.000,B 0.000,C 90.000,E1 117.513} C_DIS
LIN {X -0.064,Y -361.464,Z 1318.638,A 0.000,B 0.000,C 90.000,E1 114.823} C_DIS
LIN {X -0.121,Y -374.585,Z 1318.625,A 0.000,B 0.000,C 90.000,E1 112.461} C_DIS
LIN {X 0.018,Y -389.034,Z 1318.612,A 0.000,B 0.000,C 90.000,E1 110.120} C_DIS
LIN {X -0.123,Y -404.910,Z 1318.599,A 0.000,B 0.000,C 90.000,E1 107.873} C_DIS
LIN {X -0.128,Y -422.327,Z 1318.587,A 0.000,B 0.000,C 90.000,E1 105.662} C_DIS
LIN {X 0.107,Y -441.385,Z 1318.575,A 0.000,B 0.000,C 90.000,E1 103.480} C_DIS
LIN {X -0.005,Y -461.445,Z 1318.564,A 0.000,B 0.000,C 90.000,E1 101.478} C_DIS
LIN {X -0.006,Y -479.298,Z 1318.555,A 0.000,B 0.000,C 90.000,E1 99.849} C_DIS
LIN {X 0.005,Y -481.221,Z 1318.553,A 0.000,B 0.000,C 90.000,E1 99.613} C_DIS
LIN {X 0.014,Y -482.684,Z 1318.552,A 0.000,B 0.000,C 90.000,E1 99.378} C_DIS
LIN {X 0.179,Y -484.711,Z 1318.549,A 0.000,B 0.000,C 90.000,E1 98.859} C_DIS
LIN {X -0.124,Y -485.591,Z 1318.547,A 0.000,B 0.000,C 90.000,E1 98.398} C_DIS
LIN {X 0.134,Y -485.480,Z 1318.544,A 0.000,B 0.000,C 90.000,E1 97.871} C_DIS
LIN {X -0.153,Y -484.364,Z 1318.541,A 0.000,B 0.000,C 90.000,E1 97.409} C_DIS
LIN {X 0.154,Y -483.378,Z 1318.540,A 0.000,B 0.000,C 90.000,E1 97.125} C_DIS
LIN {X 0.040,Y -482.044,Z 1318.538,A 0.000,B 0.000,C 90.000,E1 96.891} C_DIS
LIN {X 0.120,Y -467.460,Z 1318.527,A 0.000,B 0.000,C 90.000,E1 94.878} C_DIS
LIN {X -0.118,Y -453.867,Z 1318.516,A 0.000,B 0.000,C 90.000,E1 92.865} C_DIS
LIN {X -0.004,Y -442.218,Z 1318.506,A 0.000,B 0.000,C 90.000,E1 91.031} C_DIS
LIN {X -0.135,Y -422.846,Z 1318.487,A 0.000,B 0.000,C 90.000,E1 87.593} C_DIS
LIN {X -0.185,Y -412.700,Z 1318.476,A 0.000,B 0.000,C 90.000,E1 85.698} C_DIS
LIN {X -0.003,Y -402.486,Z 1318.465,A 0.000,B 0.000,C 90.000,E1 83.742} C_DIS
LIN {X -0.013,Y -393.526,Z 1318.456,A 0.000,B 0.000,C 90.000,E1 82.064} C_DIS
LIN {X 0.153,Y -385.890,Z 1318.448,A 0.000,B 0.000,C 90.000,E1 80.622} C_DIS
LIN {X -0.025,Y -376.412,Z 1318.438,A 0.000,B 0.000,C 90.000,E1 78.926} C_DIS
LIN {X 0.002,Y -366.711,Z 1318.429,A 0.000,B 0.000,C 90.000,E1 77.173} C_DIS
LIN {X -0.071,Y -356.875,Z 1318.419,A 0.000,B 0.000,C 90.000,E1 75.408} C_DIS
LIN {X 0.121,Y -345.328,Z 1318.407,A 0.000,B 0.000,C 90.000,E1 73.268} C_DIS
LIN {X -0.061,Y -333.661,Z 1318.395,A 0.000,B 0.000,C 90.000,E1 71.148} C_DIS
LIN {X -0.097,Y -320.664,Z 1318.381,A 0.000,B 0.000,C 90.000,E1 68.646} C_DIS
LIN {X -0.076,Y -303.914,Z 1318.362,A 0.000,B 0.000,C 90.000,E1 65.101} C_DIS
LIN {X -0.089,Y -295.609,Z 1318.351,A 0.000,B 0.000,C 90.000,E1 63.127} C_DIS
LIN {X -0.141,Y -286.978,Z 1318.338,A 0.000,B 0.000,C 90.000,E1 60.795} C_DIS
LIN {X -0.020,Y -277.391,Z 1318.321,A 0.000,B 0.000,C 90.000,E1 57.709} C_DIS
LIN {X -0.154,Y -267.851,Z 1318.301,A 0.000,B 0.000,C 90.000,E1 54.276} C_DIS
LIN {X -0.130,Y -260.748,Z 1318.286,A 0.000,B 0.000,C 90.000,E1 51.457} C_DIS
LIN {X 0.075,Y -252.300,Z 1318.266,A 0.000,B 0.000,C 90.000,E1 47.838} C_DIS
LIN {X -0.024,Y -245.771,Z 1318.250,A 0.000,B 0.000,C 90.000,E1 44.960} C_DIS
LIN {X 0.011,Y -238.045,Z 1318.229,A 0.000,B 0.000,C 90.000,E1 41.272} C_DIS
LIN {X 0.062,Y -231.036,Z 1318.208,A 0.000,B 0.000,C 90.000,E1 37.523} C_DIS
LIN {X -0.140,Y -225.010,Z 1318.188,A 0.000,B 0.000,C 90.000,E1 33.785} C_DIS
LIN {X -0.031,Y -219.982,Z 1318.166,A 0.000,B 0.000,C 90.000,E1 29.922} C_DIS
LIN {X -0.084,Y -215.094,Z 1318.140,A 0.000,B 0.000,C 90.000,E1 25.283} C_DIS
LIN {X -0.074,Y -212.213,Z 1318.123,A 0.000,B 0.000,C 90.000,E1 22.153} C_DIS
LIN {X 0.091,Y -209.619,Z 1318.105,A 0.000,B 0.000,C 90.000,E1 18.960} C_DIS
LIN {X 0.063,Y -206.621,Z 1318.083,A 0.000,B 0.000,C 90.000,E1 15.009} C_DIS
LIN {X -0.113,Y -203.964,Z 1318.061,A 0.000,B 0.000,C 90.000,E1 11.074} C_DIS
LIN {X -0.092,Y -201.399,Z 1318.035,A 0.000,B 0.000,C 90.000,E1 6.258} C_DIS
LIN {X -0.037,Y -199.435,Z 1317.997,A 0.000,B 0.000,C 90.000,E1 359.542} C_DIS
LIN {X 0.049,Y -200.069,Z 1317.948,A 0.000,B 0.000,C 90.000,E1 350.622} C_DIS
LIN {X -0.085,Y -202.922,Z 1317.912,A 0.000,B 0.000,C 90.000,E1 344.212} C_DIS
LIN {X -0.025,Y -206.609,Z 1317.885,A 0.000,B 0.000,C 90.000,E1 339.390} C_DIS
LIN {X 0.005,Y -210.640,Z 1317.863,A 0.000,B 0.000,C 90.000,E1 335.409} C_DIS
LIN {X 0.039,Y -215.542,Z 1317.842,A 0.000,B 0.000,C 90.000,E1 331.463} C_DIS
LIN {X -0.010,Y -221.499,Z 1317.820,A 0.000,B 0.000,C 90.000,E1 327.582} C_DIS
LIN {X 0.126,Y -228.386,Z 1317.799,A 0.000,B 0.000,C 90.000,E1 323.703} C_DIS
LIN {X -0.095,Y -234.585,Z 1317.782,A 0.000,B 0.000,C 90.000,E1 320.723} C_DIS
LIN {X -0.107,Y -243.365,Z 1317.761,A 0.000,B 0.000,C 90.000,E1 316.986} C_DIS
LIN {X -0.026,Y -252.390,Z 1317.743,A 0.000,B 0.000,C 90.000,E1 313.662} C_DIS
LIN {X -0.081,Y -260.400,Z 1317.729,A 0.000,B 0.000,C 90.000,E1 311.148} C_DIS
LIN {X -0.109,Y -269.486,Z 1317.715,A 0.000,B 0.000,C 90.000,E1 308.669} C_DIS
LIN {X -0.160,Y -278.238,Z 1317.703,A 0.000,B 0.000,C 90.000,E1 306.583} C_DIS
LIN {X 0.157,Y -289.809,Z 1317.690,A 0.000,B 0.000,C 90.000,E1 304.119} C_DIS
LIN {X 0.007,Y -300.869,Z 1317.678,A 0.000,B 0.000,C 90.000,E1 302.133} C_DIS
LIN {X 0.129,Y -311.237,Z 1317.669,A 0.000,B 0.000,C 90.000,E1 300.463} C_DIS
LIN {X -0.020,Y -322.731,Z 1317.660,A 0.000,B 0.000,C 90.000,E1 298.871} C_DIS
LIN {X -0.066,Y -345.565,Z 1317.645,A 0.000,B 0.000,C 90.000,E1 296.052} C_DIS
LIN {X -0.030,Y -361.101,Z 1317.635,A 0.000,B 0.000,C 90.000,E1 294.259} C_DIS
LIN {X 0.050,Y -371.364,Z 1317.628,A 0.000,B 0.000,C 90.000,E1 293.078} C_DIS
LIN {X 0.135,Y -381.355,Z 1317.622,A 0.000,B 0.000,C 90.000,E1 291.897} C_DIS
LIN {X 0.131,Y -395.854,Z 1317.612,A 0.000,B 0.000,C 90.000,E1 290.174} C_DIS
LIN {X 0.036,Y -413.095,Z 1317.601,A 0.000,B 0.000,C 90.000,E1 288.236} C_DIS
LIN {X -0.055,Y -422.855,Z 1317.595,A 0.000,B 0.000,C 90.000,E1 287.149} C_DIS
LIN {X 0.098,Y -429.889,Z 1317.591,A 0.000,B 0.000,C 90.000,E1 286.315} C_DIS
LIN {X -0.106,Y -436.380,Z 1317.586,A 0.000,B 0.000,C 90.000,E1 285.536} C_DIS
LIN {X 0.060,Y -442.192,Z 1317.582,A 0.000,B 0.000,C 90.000,E1 284.717} C_DIS
LIN {X -0.041,Y -447.281,Z 1317.577,A 0.000,B 0.000,C 90.000,E1 283.939} C_DIS
LIN {X 0.235,Y -451.747,Z 1317.573,A 0.000,B 0.000,C 90.000,E1 283.119} C_DIS
LIN {X 0.110,Y -455.579,Z 1317.569,A 0.000,B 0.000,C 90.000,E1 282.355} C_DIS
LIN {X 0.196,Y -457.796,Z 1317.566,A 0.000,B 0.000,C 90.000,E1 281.827} C_DIS
LIN {X -0.246,Y -459.749,Z 1317.563,A 0.000,B 0.000,C 90.000,E1 281.366} C_DIS
LIN {X -0.141,Y -461.302,Z 1317.560,A 0.000,B 0.000,C 90.000,E1 280.838} C_DIS
LIN {X -0.026,Y -462.523,Z 1317.557,A 0.000,B 0.000,C 90.000,E1 280.310} C_DIS
LIN {X 0.017,Y -463.310,Z 1317.554,A 0.000,B 0.000,C 90.000,E1 279.792} C_DIS
LIN {X 0.147,Y -463.646,Z 1317.552,A 0.000,B 0.000,C 90.000,E1 279.265} C_DIS
LIN {X 0.206,Y -463.551,Z 1317.549,A 0.000,B 0.000,C 90.000,E1 278.746} C_DIS
LIN {X -0.123,Y -463.001,Z 1317.546,A 0.000,B 0.000,C 90.000,E1 278.276} C_DIS
LIN {X -0.061,Y -462.025,Z 1317.543,A 0.000,B 0.000,C 90.000,E1 277.757} C_DIS
LIN {X -0.001,Y -460.551,Z 1317.540,A 0.000,B 0.000,C 90.000,E1 277.239} C_DIS
LIN {X 0.053,Y -458.554,Z 1317.537,A 0.000,B 0.000,C 90.000,E1 276.720} C_DIS
LIN {X 0.100,Y -456.073,Z 1317.535,A 0.000,B 0.000,C 90.000,E1 276.201} C_DIS
LIN {X 0.127,Y -452.983,Z 1317.532,A 0.000,B 0.000,C 90.000,E1 275.682} C_DIS
LIN {X 0.138,Y -449.356,Z 1317.529,A 0.000,B 0.000,C 90.000,E1 275.163} C_DIS
LIN {X 0.126,Y -444.942,Z 1317.526,A 0.000,B 0.000,C 90.000,E1 274.645} C_DIS
LIN {X 0.059,Y -439.587,Z 1317.523,A 0.000,B 0.000,C 90.000,E1 274.131} C_DIS
LIN {X -0.121,Y -433.658,Z 1317.520,A 0.000,B 0.000,C 90.000,E1 273.669} C_DIS
LIN {X 0.078,Y -427.307,Z 1317.518,A 0.000,B 0.000,C 90.000,E1 273.212} C_DIS
LIN {X -0.139,Y -420.728,Z 1317.516,A 0.000,B 0.000,C 90.000,E1 272.865} C_DIS
LIN {X 0.025,Y -414.036,Z 1317.514,A 0.000,B 0.000,C 90.000,E1 272.522} C_DIS
LIN {X 0.076,Y -407.134,Z 1317.512,A 0.000,B 0.000,C 90.000,E1 272.236} C_DIS
LIN {X 0.024,Y -399.946,Z 1317.511,A 0.000,B 0.000,C 90.000,E1 272.007} C_DIS
LIN {X -0.150,Y -392.607,Z 1317.510,A 0.000,B 0.000,C 90.000,E1 271.835} C_DIS
LIN {X -0.082,Y -385.032,Z 1317.509,A 0.000,B 0.000,C 90.000,E1 271.661} C_DIS
LIN {X 0.186,Y -376.997,Z 1317.508,A 0.000,B 0.000,C 90.000,E1 271.489} C_DIS
LIN {X 0.127,Y -363.158,Z 1317.508,A 0.000,B 0.000,C 90.000,E1 271.375} C_DIS
LIN {X -0.158,Y -347.546,Z 1317.507,A 0.000,B 0.000,C 90.000,E1 271.375} C_DIS
LIN {X 0.069,Y -181.383,Z 1317.507,A 0.000,B 0.000,C 90.000,E1 271.318} C_DIS
LIN {X -0.067,Y -181.580,Z 1317.502,A 0.000,B 0.000,C 90.000,E1 270.344} C_DIS
LIN {X -0.062,Y -180.882,Z 1317.473,A 0.000,B 0.000,C 90.000,E1 265.122} C_DIS
LIN {X -0.003,Y -179.002,Z 1317.445,A 0.000,B 0.000,C 90.000,E1 260.038} C_DIS
LIN {X 0.091,Y -178.601,Z 1317.440,A 0.000,B 0.000,C 90.000,E1 259.162} C_DIS
LIN {X -0.015,Y -175.653,Z 1317.412,A 0.000,B 0.000,C 90.000,E1 254.102} C_DIS
LIN {X -0.010,Y -172.370,Z 1317.388,A 0.000,B 0.000,C 90.000,E1 249.826} C_DIS
LIN {X 0.005,Y -171.164,Z 1317.378,A 0.000,B 0.000,C 90.000,E1 248.103} C_DIS
LIN {X 0.048,Y -167.462,Z 1317.354,A 0.000,B 0.000,C 90.000,E1 243.768} C_DIS
LIN {X -0.019,Y -166.858,Z 1317.349,A 0.000,B 0.000,C 90.000,E1 242.922} C_DIS
LIN {X 0.046,Y -162.843,Z 1317.325,A 0.000,B 0.000,C 90.000,E1 238.535} C_DIS
LIN {X 0.022,Y -161.527,Z 1317.316,A 0.000,B 0.000,C 90.000,E1 236.786} C_DIS
LIN {X 0.061,Y -157.527,Z 1317.291,A 0.000,B 0.000,C 90.000,E1 232.351} C_DIS
LIN {X -0.006,Y -155.552,Z 1317.276,A 0.000,B 0.000,C 90.000,E1 229.703} C_DIS
LIN {X -0.072,Y -151.844,Z 1317.251,A 0.000,B 0.000,C 90.000,E1 225.243} C_DIS
LIN {X -0.058,Y -150.062,Z 1317.236,A 0.000,B 0.000,C 90.000,E1 222.528} C_DIS
LIN {X -0.023,Y -146.872,Z 1317.211,A 0.000,B 0.000,C 90.000,E1 217.971} C_DIS
LIN {X -0.033,Y -145.457,Z 1317.196,A 0.000,B 0.000,C 90.000,E1 215.231} C_DIS
LIN {X 0.080,Y -142.872,Z 1317.170,A 0.000,B 0.000,C 90.000,E1 210.590} C_DIS
LIN {X 0.005,Y -141.490,Z 1317.150,A 0.000,B 0.000,C 90.000,E1 206.924} C_DIS
LIN {X -0.010,Y -139.385,Z 1317.114,A 0.000,B 0.000,C 90.000,E1 200.429} C_DIS
LIN {X -0.021,Y -138.840,Z 1317.098,A 0.000,B 0.000,C 90.000,E1 197.638} C_DIS
LIN {X 0.039,Y -138.353,Z 1317.056,A 0.000,B 0.000,C 90.000,E1 190.141} C_DIS
LIN {X 0.035,Y -139.520,Z 1317.005,A 0.000,B 0.000,C 90.000,E1 180.802} C_DIS
LIN {X -0.024,Y -141.182,Z 1316.974,A 0.000,B 0.000,C 90.000,E1 175.241} C_DIS
LIN {X -0.054,Y -142.561,Z 1316.958,A 0.000,B 0.000,C 90.000,E1 172.470} C_DIS
LIN {X 0.013,Y -144.842,Z 1316.932,A 0.000,B 0.000,C 90.000,E1 167.825} C_DIS
LIN {X -0.001,Y -147.466,Z 1316.912,A 0.000,B 0.000,C 90.000,E1 164.157} C_DIS
LIN {X 0.026,Y -150.050,Z 1316.892,A 0.000,B 0.000,C 90.000,E1 160.496} C_DIS
LIN {X 0.030,Y -153.393,Z 1316.872,A 0.000,B 0.000,C 90.000,E1 156.869} C_DIS
LIN {X 0.078,Y -155.924,Z 1316.857,A 0.000,B 0.000,C 90.000,E1 154.152} C_DIS
LIN {X 0.052,Y -159.790,Z 1316.837,A 0.000,B 0.000,C 90.000,E1 150.589} C_DIS
LIN {X 0.038,Y -162.030,Z 1316.827,A 0.000,B 0.000,C 90.000,E1 148.820} C_DIS
LIN {X 0.012,Y -166.226,Z 1316.807,A 0.000,B 0.000,C 90.000,E1 145.308} C_DIS
LIN {X 0.013,Y -171.242,Z 1316.788,A 0.000,B 0.000,C 90.000,E1 141.823} C_DIS
LIN {X -0.064,Y -176.129,Z 1316.769,A 0.000,B 0.000,C 90.000,E1 138.405} C_DIS
LIN {X 0.052,Y -180.396,Z 1316.755,A 0.000,B 0.000,C 90.000,E1 135.810} C_DIS
LIN {X 0.029,Y -185.804,Z 1316.736,A 0.000,B 0.000,C 90.000,E1 132.447} C_DIS
LIN {X 0.083,Y -190.422,Z 1316.722,A 0.000,B 0.000,C 90.000,E1 129.930} C_DIS
LIN {X -0.024,Y -197.746,Z 1316.699,A 0.000,B 0.000,C 90.000,E1 125.851} C_DIS
LIN {X -0.108,Y -199.288,Z 1316.695,A 0.000,B 0.000,C 90.000,E1 125.105} C_DIS
LIN {X -0.203,Y -308.717,Z 1316.695,A 0.000,B 0.000,C 90.000,E1 125.105} C_DIS
LIN {X 0.023,Y -310.995,Z 1316.695,A 0.000,B 0.000,C 90.000,E1 125.025} C_DIS
LIN {X 0.065,Y -313.906,Z 1316.694,A 0.000,B 0.000,C 90.000,E1 124.898} C_DIS
LIN {X -0.025,Y -317.368,Z 1316.693,A 0.000,B 0.000,C 90.000,E1 124.659} C_DIS
LIN {X 0.104,Y -321.005,Z 1316.690,A 0.000,B 0.000,C 90.000,E1 124.199} C_DIS
LIN {X -0.085,Y -322.860,Z 1316.688,A 0.000,B 0.000,C 90.000,E1 123.913} C_DIS
LIN {X -0.006,Y -324.301,Z 1316.687,A 0.000,B 0.000,C 90.000,E1 123.579} C_DIS
LIN {X -0.080,Y -337.121,Z 1316.667,A 0.000,B 0.000,C 90.000,E1 120.129} C_DIS
LIN {X 0.030,Y -349.059,Z 1316.652,A 0.000,B 0.000,C 90.000,E1 117.334} C_DIS
LIN {X -0.146,Y -362.452,Z 1316.637,A 0.000,B 0.000,C 90.000,E1 114.643} C_DIS
LIN {X -0.033,Y -375.676,Z 1316.624,A 0.000,B 0.000,C 90.000,E1 112.259} C_DIS
LIN {X -0.007,Y -390.235,Z 1316.611,A 0.000,B 0.000,C 90.000,E1 109.939} C_DIS
LIN {X -0.119,Y -406.232,Z 1316.598,A 0.000,B 0.000,C 90.000,E1 107.692} C_DIS
LIN {X -0.092,Y -423.778,Z 1316.586,A 0.000,B 0.000,C 90.000,E1 105.481} C_DIS
LIN {X 0.187,Y -442.963,Z 1316.574,A 0.000,B 0.000,C 90.000,E1 103.300} C_DIS
LIN {X 0.185,Y -463.070,Z 1316.563,A 0.000,B 0.000,C 90.000,E1 101.299} C_DIS
LIN {X 0.189,Y -478.465,Z 1316.555,A 0.000,B 0.000,C 90.000,E1 99.905} C_DIS
LIN {X -0.195,Y -480.493,Z 1316.554,A 0.000,B 0.000,C 90.000,E1 99.726} C_DIS
LIN {X 0.075,Y -482.192,Z 1316.552,A 0.000,B 0.000,C 90.000,E1 99.443} C_DIS
LIN {X -0.049,Y -483.465,Z 1316.551,A 0.000,B 0.000,C 90.000,E1 99.208} C_DIS
LIN {X 0.125,Y -485.034,Z 1316.548,A 0.000,B 0.000,C 90.000,E1 98.690} C_DIS
LIN {X -0.103,Y -485.540,Z 1316.546,A 0.000,B 0.000,C 90.000,E1 98.219} C_DIS
LIN {X 0.088,Y -485.066,Z 1316.543,A 0.000,B 0.000,C 90.000,E1 97.701} C_DIS
LIN {X -0.198,Y -483.542,Z 1316.540,A 0.000,B 0.000,C 90.000,E1 97.239} C_DIS
LIN {X 0.167,Y -482.306,Z 1316.539,A 0.000,B 0.000,C 90.000,E1 96.947} C_DIS
LIN {X -0.005,Y -480.655,Z 1316.537,A 0.000,B 0.000,C 90.000,E1 96.720} C_DIS
LIN {X -0.018,Y -469.494,Z 1316.529,A 0.000,B 0.000,C 90.000,E1 95.220} C_DIS
LIN {X 0.013,Y -454.142,Z 1316.516,A 0.000,B 0.000,C 90.000,E1 92.922} C_DIS
LIN {X 0.134,Y -442.441,Z 1316.506,A 0.000,B 0.000,C 90.000,E1 91.088} C_DIS
LIN {X 0.000,Y -423.048,Z 1316.487,A 0.000,B 0.000,C 90.000,E1 87.650} C_DIS
LIN {X -0.045,Y -412.893,Z 1316.476,A 0.000,B 0.000,C 90.000,E1 85.755} C_DIS
LIN {X 0.135,Y -402.693,Z 1316.466,A 0.000,B 0.000,C 90.000,E1 83.799} C_DIS
LIN {X 0.074,Y -393.751,Z 1316.456,A 0.000,B 0.000,C 90.000,E1 82.129} C_DIS
LIN {X -0.081,Y -386.157,Z 1316.448,A 0.000,B 0.000,C 90.000,E1 80.735} C_DIS
LIN {X 0.052,Y -376.686,Z 1316.439,A 0.000,B 0.000,C 90.000,E1 78.993} C_DIS
LIN {X 0.156,Y -366.987,Z 1316.429,A 0.000,B 0.000,C 90.000,E1 77.229} C_DIS
LIN {X 0.086,Y -357.156,Z 1316.419,A 0.000,B 0.000,C 90.000,E1 75.463} C_DIS
LIN {X -0.053,Y -345.600,Z 1316.408,A 0.000,B 0.000,C 90.000,E1 73.378} C_DIS
LIN {X -0.003,Y -333.946,Z 1316.396,A 0.000,B 0.000,C 90.000,E1 71.221} C_DIS
LIN {X -0.043,Y -320.921,Z 1316.382,A 0.000,B 0.000,C 90.000,E1 68.720} C_DIS
LIN {X -0.031,Y -304.170,Z 1316.362,A 0.000,B 0.000,C 90.000,E1 65.177} C_DIS
LIN {X -0.038,Y -294.553,Z 1316.349,A 0.000,B 0.000,C 90.000,E1 62.871} C_DIS
LIN {X 0.046,Y -287.208,Z 1316.338,A 0.000,B 0.000,C 90.000,E1 60.845} C_DIS
LIN {X 0.069,Y -278.629,Z 1316.323,A 0.000,B 0.000,C 90.000,E1 58.122} C_DIS
LIN {X -0.030,Y -268.973,Z 1316.304,A 0.000,B 0.000,C 90.000,E1 54.689} C_DIS
LIN {X -0.023,Y -260.090,Z 1316.284,A 0.000,B 0.000,C 90.000,E1 51.170} C_DIS
LIN {X -0.070,Y -253.318,Z 1316.268,A 0.000,B 0.000,C 90.000,E1 48.324} C_DIS
LIN {X 0.032,Y -246.768,Z 1316.252,A 0.000,B 0.000,C 90.000,E1 45.405} C_DIS
LIN {X -0.069,Y -238.952,Z 1316.232,A 0.000,B 0.000,C 90.000,E1 41.757} C_DIS
LIN {X -0.019,Y -231.831,Z 1316.211,A 0.000,B 0.000,C 90.000,E1 38.016} C_DIS
LIN {X 0.115,Y -225.650,Z 1316.190,A 0.000,B 0.000,C 90.000,E1 34.199} C_DIS
LIN {X 0.052,Y -220.502,Z 1316.169,A 0.000,B 0.000,C 90.000,E1 30.384} C_DIS
LIN {X 0.112,Y -215.465,Z 1316.143,A 0.000,B 0.000,C 90.000,E1 25.720} C_DIS
LIN {X -0.020,Y -211.838,Z 1316.121,A 0.000,B 0.000,C 90.000,E1 21.844} C_DIS
LIN {X 0.090,Y -208.588,Z 1316.099,A 0.000,B 0.000,C 90.000,E1 17.873} C_DIS
LIN {X -0.031,Y -205.666,Z 1316.077,A 0.000,B 0.000,C 90.000,E1 13.939} C_DIS
LIN {X 0.047,Y -203.572,Z 1316.060,A 0.000,B 0.000,C 90.000,E1 10.725} C_DIS
LIN {X 0.050,Y -201.061,Z 1316.033,A 0.000,B 0.000,C 90.000,E1 5.910} C_DIS
LIN {X -0.036,Y -199.266,Z 1315.997,A 0.000,B 0.000,C 90.000,E1 359.542} C_DIS
LIN {X 0.038,Y -199.963,Z 1315.948,A 0.000,B 0.000,C 90.000,E1 350.622} C_DIS
LIN {X 0.096,Y -202.900,Z 1315.912,A 0.000,B 0.000,C 90.000,E1 344.157} C_DIS
LIN {X -0.041,Y -206.638,Z 1315.885,A 0.000,B 0.000,C 90.000,E1 339.390} C_DIS
LIN {X -0.010,Y -210.707,Z 1315.863,A 0.000,B 0.000,C 90.000,E1 335.409} C_DIS
LIN {X 0.027,Y -215.627,Z 1315.842,A 0.000,B 0.000,C 90.000,E1 331.463} C_DIS
LIN {X -0.020,Y -221.586,Z 1315.820,A 0.000,B 0.000,C 90.000,E1 327.582} C_DIS
LIN {X 0.119,Y -228.481,Z 1315.798,A 0.000,B 0.000,C 90.000,E1 323.703} C_DIS
LIN {X -0.100,Y -234.675,Z 1315.782,A 0.000,B 0.000,C 90.000,E1 320.723} C_DIS
LIN {X 0.068,Y -243.431,Z 1315.761,A 0.000,B 0.000,C 90.000,E1 316.944} C_DIS
LIN {X -0.027,Y -252.468,Z 1315.743,A 0.000,B 0.000,C 90.000,E1 313.662} C_DIS
LIN {X -0.080,Y -260.450,Z 1315.729,A 0.000,B 0.000,C 90.000,E1 311.148} C_DIS
LIN {X -0.106,Y -269.540,Z 1315.715,A 0.000,B 0.000,C 90.000,E1 308.669} C_DIS
LIN {X -0.157,Y -278.297,Z 1315.703,A 0.000,B 0.000,C 90.000,E1 306.583} C_DIS
LIN {X 0.162,Y -289.852,Z 1315.690,A 0.000,B 0.000,C 90.000,E1 304.119} C_DIS
LIN {X 0.014,Y -300.932,Z 1315.679,A 0.000,B 0.000,C 90.000,E1 302.133} C_DIS
LIN {X 0.095,Y -309.153,Z 1315.671,A 0.000,B 0.000,C 90.000,E1 300.797} C_DIS
LIN {X -0.079,Y -320.380,Z 1315.662,A 0.000,B 0.000,C 90.000,E1 299.205} C_DIS
LIN {X -0.072,Y -342.974,Z 1315.646,A 0.000,B 0.000,C 90.000,E1 296.360} C_DIS
LIN {X 0.021,Y -356.123,Z 1315.638,A 0.000,B 0.000,C 90.000,E1 294.823} C_DIS
LIN {X 0.022,Y -369.151,Z 1315.630,A 0.000,B 0.000,C 90.000,E1 293.334} C_DIS
LIN {X -0.172,Y -381.745,Z 1315.621,A 0.000,B 0.000,C 90.000,E1 291.897} C_DIS
LIN {X -0.138,Y -398.650,Z 1315.610,A 0.000,B 0.000,C 90.000,E1 289.885} C_DIS
LIN {X -0.123,Y -416.086,Z 1315.599,A 0.000,B 0.000,C 90.000,E1 287.928} C_DIS
LIN {X -0.045,Y -428.077,Z 1315.592,A 0.000,B 0.000,C 90.000,E1 286.551} C_DIS
LIN {X 0.158,Y -434.703,Z 1315.587,A 0.000,B 0.000,C 90.000,E1 285.717} C_DIS
LIN {X -0.121,Y -440.685,Z 1315.583,A 0.000,B 0.000,C 90.000,E1 284.954} C_DIS
LIN {X 0.202,Y -445.959,Z 1315.579,A 0.000,B 0.000,C 90.000,E1 284.120} C_DIS
LIN {X 0.026,Y -450.499,Z 1315.574,A 0.000,B 0.000,C 90.000,E1 283.355} C_DIS
LIN {X -0.106,Y -454.530,Z 1315.570,A 0.000,B 0.000,C 90.000,E1 282.591} C_DIS
LIN {X -0.210,Y -457.961,Z 1315.566,A 0.000,B 0.000,C 90.000,E1 281.827} C_DIS
LIN {X -0.111,Y -459.873,Z 1315.563,A 0.000,B 0.000,C 90.000,E1 281.299} C_DIS
LIN {X -0.094,Y -461.463,Z 1315.560,A 0.000,B 0.000,C 90.000,E1 280.782} C_DIS
LIN {X 0.023,Y -462.640,Z 1315.557,A 0.000,B 0.000,C 90.000,E1 280.254} C_DIS
LIN {X 0.146,Y -463.396,Z 1315.554,A 0.000,B 0.000,C 90.000,E1 279.726} C_DIS
LIN {X 0.198,Y -463.748,Z 1315.551,A 0.000,B 0.000,C 90.000,E1 279.208} C_DIS
LIN {X -0.200,Y -463.637,Z 1315.548,A 0.000,B 0.000,C 90.000,E1 278.746} C_DIS
LIN {X -0.068,Y -463.125,Z 1315.546,A 0.000,B 0.000,C 90.000,E1 278.219} C_DIS
LIN {X -0.006,Y -462.131,Z 1315.543,A 0.000,B 0.000,C 90.000,E1 277.701} C_DIS
LIN {X 0.055,Y -460.644,Z 1315.540,A 0.000,B 0.000,C 90.000,E1 277.182} C_DIS
LIN {X 0.110,Y -458.642,Z 1315.537,A 0.000,B 0.000,C 90.000,E1 276.663} C_DIS
LIN {X 0.157,Y -456.142,Z 1315.534,A 0.000,B 0.000,C 90.000,E1 276.144} C_DIS
LIN {X 0.185,Y -453.066,Z 1315.531,A 0.000,B 0.000,C 90.000,E1 275.625} C_DIS
LIN {X 0.195,Y -449.428,Z 1315.529,A 0.000,B 0.000,C 90.000,E1 275.106} C_DIS
LIN {X 0.185,Y -445.002,Z 1315.526,A 0.000,B 0.000,C 90.000,E1 274.588} C_DIS
LIN {X 0.118,Y -439.695,Z 1315.523,A 0.000,B 0.000,C 90.000,E1 274.073} C_DIS
LIN {X -0.068,Y -433.695,Z 1315.520,A 0.000,B 0.000,C 90.000,E1 273.612} C_DIS
LIN {X 0.164,Y -427.402,Z 1315.518,A 0.000,B 0.000,C 90.000,E1 273.154} C_DIS
LIN {X -0.048,Y -420.860,Z 1315.516,A 0.000,B 0.000,C 90.000,E1 272.808} C_DIS
LIN {X 0.065,Y -414.013,Z 1315.514,A 0.000,B 0.000,C 90.000,E1 272.465} C_DIS
LIN {X 0.106,Y -406.882,Z 1315.512,A 0.000,B 0.000,C 90.000,E1 272.178} C_DIS
LIN {X 0.093,Y -399.753,Z 1315.511,A 0.000,B 0.000,C 90.000,E1 271.949} C_DIS
LIN {X 0.194,Y -389.035,Z 1315.509,A 0.000,B 0.000,C 90.000,E1 271.661} C_DIS
LIN {X -0.007,Y -381.166,Z 1315.509,A 0.000,B 0.000,C 90.000,E1 271.547} C_DIS
LIN {X 0.004,Y -372.253,Z 1315.508,A 0.000,B 0.000,C 90.000,E1 271.432} C_DIS
LIN {X 0.175,Y -358.242,Z 1315.507,A 0.000,B 0.000,C 90.000,E1 271.318} C_DIS
LIN {X 0.060,Y -351.855,Z 1315.507,A 0.000,B 0.000,C 90.000,E1 271.318} C_DIS
LIN {X 0.002,Y -181.387,Z 1315.507,A 0.000,B 0.000,C 90.000,E1 271.318} C_DIS
LIN {X 0.045,Y -181.580,Z 1315.502,A 0.000,B 0.000,C 90.000,E1 270.286} C_DIS
LIN {X 0.049,Y -180.878,Z 1315.473,A 0.000,B 0.000,C 90.000,E1 265.065} C_DIS
LIN {X -0.071,Y -178.997,Z 1315.445,A 0.000,B 0.000,C 90.000,E1 260.038} C_DIS
LIN {X 0.024,Y -178.585,Z 1315.440,A 0.000,B 0.000,C 90.000,E1 259.162} C_DIS
LIN {X -0.083,Y -175.637,Z 1315.411,A 0.000,B 0.000,C 90.000,E1 254.102} C_DIS
LIN {X -0.016,Y -172.356,Z 1315.388,A 0.000,B 0.000,C 90.000,E1 249.806} C_DIS
LIN {X -0.061,Y -171.142,Z 1315.378,A 0.000,B 0.000,C 90.000,E1 248.103} C_DIS
LIN {X -0.017,Y -167.445,Z 1315.354,A 0.000,B 0.000,C 90.000,E1 243.768} C_DIS
LIN {X 0.065,Y -166.841,Z 1315.349,A 0.000,B 0.000,C 90.000,E1 242.871} C_DIS
LIN {X -0.017,Y -162.826,Z 1315.325,A 0.000,B 0.000,C 90.000,E1 238.535} C_DIS
LIN {X 0.046,Y -161.511,Z 1315.315,A 0.000,B 0.000,C 90.000,E1 236.755} C_DIS
LIN {X -0.001,Y -157.509,Z 1315.291,A 0.000,B 0.000,C 90.000,E1 232.351} C_DIS
LIN {X 0.033,Y -155.531,Z 1315.276,A 0.000,B 0.000,C 90.000,E1 229.666} C_DIS
LIN {X 0.082,Y -151.827,Z 1315.251,A 0.000,B 0.000,C 90.000,E1 225.162} C_DIS
LIN {X -0.007,Y -150.043,Z 1315.236,A 0.000,B 0.000,C 90.000,E1 222.486} C_DIS
LIN {X 0.008,Y -146.858,Z 1315.211,A 0.000,B 0.000,C 90.000,E1 217.935} C_DIS
LIN {X 0.025,Y -145.442,Z 1315.196,A 0.000,B 0.000,C 90.000,E1 215.185} C_DIS
LIN {X 0.021,Y -142.862,Z 1315.170,A 0.000,B 0.000,C 90.000,E1 210.590} C_DIS
LIN {X 0.073,Y -141.478,Z 1315.149,A 0.000,B 0.000,C 90.000,E1 206.873} C_DIS
LIN {X -0.068,Y -139.381,Z 1315.113,A 0.000,B 0.000,C 90.000,E1 200.429} C_DIS
LIN {X 0.053,Y -138.834,Z 1315.098,A 0.000,B 0.000,C 90.000,E1 197.583} C_DIS
LIN {X -0.019,Y -138.353,Z 1315.056,A 0.000,B 0.000,C 90.000,E1 190.141} C_DIS
LIN {X -0.023,Y -139.524,Z 1315.004,A 0.000,B 0.000,C 90.000,E1 180.802} C_DIS
LIN {X 0.057,Y -141.193,Z 1314.973,A 0.000,B 0.000,C 90.000,E1 175.184} C_DIS
LIN {X 0.029,Y -142.569,Z 1314.958,A 0.000,B 0.000,C 90.000,E1 172.413} C_DIS
LIN {X -0.016,Y -144.857,Z 1314.932,A 0.000,B 0.000,C 90.000,E1 167.813} C_DIS
LIN {X -0.061,Y -147.482,Z 1314.912,A 0.000,B 0.000,C 90.000,E1 164.157} C_DIS
LIN {X -0.035,Y -150.069,Z 1314.892,A 0.000,B 0.000,C 90.000,E1 160.496} C_DIS
LIN {X -0.031,Y -153.417,Z 1314.871,A 0.000,B 0.000,C 90.000,E1 156.869} C_DIS
LIN {X 0.016,Y -156.838,Z 1314.851,A 0.000,B 0.000,C 90.000,E1 153.256} C_DIS
LIN {X 0.088,Y -160.917,Z 1314.832,A 0.000,B 0.000,C 90.000,E1 149.665} C_DIS
LIN {X 0.032,Y -163.042,Z 1314.822,A 0.000,B 0.000,C 90.000,E1 147.916} C_DIS
LIN {X 0.038,Y -167.434,Z 1314.802,A 0.000,B 0.000,C 90.000,E1 144.402} C_DIS
LIN {X -0.052,Y -171.272,Z 1314.788,A 0.000,B 0.000,C 90.000,E1 141.823} C_DIS
LIN {X -0.014,Y -176.163,Z 1314.769,A 0.000,B 0.000,C 90.000,E1 138.366} C_DIS
LIN {X -0.016,Y -180.435,Z 1314.755,A 0.000,B 0.000,C 90.000,E1 135.810} C_DIS
LIN {X -0.041,Y -185.840,Z 1314.736,A 0.000,B 0.000,C 90.000,E1 132.447} C_DIS
LIN {X 0.012,Y -190.463,Z 1314.722,A 0.000,B 0.000,C 90.000,E1 129.930} C_DIS
LIN {X -0.082,Y -196.215,Z 1314.704,A 0.000,B 0.000,C 90.000,E1 126.664} C_DIS
LIN {X 0.124,Y -199.314,Z 1314.695,A 0.000,B 0.000,C 90.000,E1 125.025} C_DIS
LIN {X 0.157,Y -309.132,Z 1314.695,A 0.000,B 0.000,C 90.000,E1 125.025} C_DIS
LIN {X -0.090,Y -311.388,Z 1314.694,A 0.000,B 0.000,C 90.000,E1 125.025} C_DIS
LIN {X -0.035,Y -314.619,Z 1314.694,A 0.000,B 0.000,C 90.000,E1 124.865} C_DIS
LIN {X 0.043,Y -318.113,Z 1314.692,A 0.000,B 0.000,C 90.000,E1 124.565} C_DIS
LIN {X -0.139,Y -321.730,Z 1314.689,A 0.000,B 0.000,C 90.000,E1 124.119} C_DIS
LIN {X -0.064,Y -323.427,Z 1314.688,A 0.000,B 0.000,C 90.000,E1 123.785} C_DIS
LIN {X -0.168,Y -325.846,Z 1314.684,A 0.000,B 0.000,C 90.000,E1 123.166} C_DIS
LIN {X -0.179,Y -336.342,Z 1314.668,A 0.000,B 0.000,C 90.000,E1 120.335} C_DIS
LIN {X 0.075,Y -348.183,Z 1314.653,A 0.000,B 0.000,C 90.000,E1 117.513} C_DIS
LIN {X 0.193,Y -361.477,Z 1314.638,A 0.000,B 0.000,C 90.000,E1 114.771} C_DIS
LIN {X -0.194,Y -374.603,Z 1314.625,A 0.000,B 0.000,C 90.000,E1 112.461} C_DIS
LIN {X -0.057,Y -389.057,Z 1314.612,A 0.000,B 0.000,C 90.000,E1 110.120} C_DIS
LIN {X 0.184,Y -404.941,Z 1314.599,A 0.000,B 0.000,C 90.000,E1 107.819} C_DIS
LIN {X 0.198,Y -422.365,Z 1314.587,A 0.000,B 0.000,C 90.000,E1 105.607} C_DIS
LIN {X 0.014,Y -441.442,Z 1314.575,A 0.000,B 0.000,C 90.000,E1 103.480} C_DIS
LIN {X -0.095,Y -461.505,Z 1314.564,A 0.000,B 0.000,C 90.000,E1 101.478} C_DIS
LIN {X -0.088,Y -476.913,Z 1314.556,A 0.000,B 0.000,C 90.000,E1 100.074} C_DIS
LIN {X -0.075,Y -479.279,Z 1314.555,A 0.000,B 0.000,C 90.000,E1 99.849} C_DIS
LIN {X 0.021,Y -481.074,Z 1314.553,A 0.000,B 0.000,C 90.000,E1 99.613} C_DIS
LIN {X -0.101,Y -482.596,Z 1314.552,A 0.000,B 0.000,C 90.000,E1 99.378} C_DIS
LIN {X 0.175,Y -483.732,Z 1314.551,A 0.000,B 0.000,C 90.000,E1 99.095} C_DIS
LIN {X -0.054,Y -485.084,Z 1314.548,A 0.000,B 0.000,C 90.000,E1 98.624} C_DIS
